METHOD PUBLIC Pop : T_PTR_STRUCT
// Remove a paper from the buffer
VAR_INPUT
END_VAR
Pop.eStatus := E_PTR_Status.Gone;
Pop.lrePositionOnBelt_mm := 0.0;
Pop.lrePositionOnBeltAdjusted_mm := 0.0;
Pop.udiItemId := 0;
Pop.udiTimeOnBelt_us := 0;


IF m_intPaperOnBelt > 0 THEN
	Pop := m_arBuffer[m_intFirstPaperIdx];
	m_arBuffer[m_intFirstPaperIdx].udiItemId := 0;
	m_arBuffer[m_intFirstPaperIdx].lrePositionOnBelt_mm := 0.0;
	m_arBuffer[m_intFirstPaperIdx].lrePositionOnBeltAdjusted_mm := 0.0;
	m_arBuffer[m_intFirstPaperIdx].udiTimeOnBelt_us := 0;
	m_arBuffer[m_intFirstPaperIdx].eStatus := E_PTR_Status.Gone;
	m_intPaperOnBelt := m_intPaperOnBelt - 1;

	IF m_intPaperOnBelt = 0 THEN
		m_arPositionList[0] := m_arBuffer[m_intFirstPaperIdx];
	END_IF

	m_intFirstPaperIdx := (m_intFirstPaperIdx + 1) MOD THIS^.cMAXBUFFERSIZE;
END_IF
END_METHOD

PROPERTY PUBLIC PositionList : POINTER TO T_PTR_STRUCT
GET
VAR
	iIdx			: INT;
	iNdx			: INT;
END_VAR
PositionList := ADR(m_arPositionList);
END_GET
SET
END_SET
END_PROPERTY

METHOD PUBLIC Push : BOOL
// Add (Push) a paper into the buffer
// Return an ID for the paper
VAR_INPUT
	In_udiItemId			: UDINT;
END_VAR
Push := FALSE;

IF m_intPaperOnBelt < THIS^.cMAXBUFFERSIZE THEN
	m_intLastPaperIdx := (m_intLastPaperIdx + 1) MOD THIS^.cMAXBUFFERSIZE;
	m_arBuffer[m_intLastPaperIdx].udiItemId := In_udiItemId;
	m_arBuffer[m_intLastPaperIdx].lrePositionOnBelt_mm := 0.0;
	m_arBuffer[m_intLastPaperIdx].lrePositionOnBeltAdjusted_mm := 0.0;
	m_arBuffer[m_intLastPaperIdx].udiTimeOnBelt_us := 0;
	m_arBuffer[m_intLastPaperIdx].eStatus := E_PTR_Status.EnterBusy;
	m_intPaperOnBelt := m_intPaperOnBelt + 1;
	Push := TRUE;
END_IF
END_METHOD

METHOD PUBLIC Reset : BOOL
VAR_INPUT
END_VAR
m_intFirstPaperIdx := 0;
m_intLastPaperIdx := -1;
m_intPaperOnBelt := 0;
END_METHOD

PROPERTY PUBLIC TimeBase : UDINT
GET
TimeBase := m_udiTimeBase_us;
END_GET
SET
m_udiTimeBase_us := TimeBase;
END_SET
END_PROPERTY

END_FUNCTION_BLOCK

// POUs/Controller/Driver/TCP (TCP communication driver)/FB_TCP
FUNCTION_BLOCK FB_TCP EXTENDS FB_CtrlBase
VAR
	/// Specific interface struct for public access
	SIf: T_Ctrl_SIf_TCP;
	intSendState: INT := 0;
	fbClientConnection: TC2_TCPIP.FB_ClientServerConnection;
	fbSend: TC2_TCPIP.FB_SocketSend;
	fbRecieve: TC2_TCPIP.FB_SocketReceive;
	/// buffer for recieved messages
	fbRecieveBuffer: FB_DataSetFifo;
	/// buffer for messages to be sendt
	fbSendBuffer: FB_DataSetFifo;
	stNextHead: ST_Header;
	bRecievedAck: BOOL;
	bRecievedNack: BOOL;
	iSendSize: UDINT;
	iNumSendTry: INT;
	tonSendTime: TON;
	pSendHeader: POINTER TO ST_Header;
	pByteSend: POINTER TO ARRAY[0..MAX_DATASET_SIZE] OF BYTE;
	pRecieveHead: POINTER TO ST_Header;
	pByteReceive: POINTER TO ARRAY[0..MAX_DATASET_SIZE] OF BYTE;
	naRecieveData: ARRAY[0..MAX_DATASET_SIZE] OF BYTE;
	pRecieveData: POINTER TO ARRAY[0..MAX_DATASET_SIZE] OF BYTE;
END_VAR
VAR CONSTANT
	cSendIdle: INT := 0;
	cSendBusy: INT := 1;
	cSendWait: INT := 2;
END_VAR

(*__________________________________________________________________________________________________
¦	
¦	Vistaprint Schweiz GmbH
¦	CH - 8401 Winterthur
¦
¦	www.vistaprint.ch - info@vistaprint.ch
¦___________________________________________________________________________________________________

Function desription:



History:
Version		Date			Author		Comment
---------------------------------------------------------------------------------------------------
0.00.1		21.05.2014		AVME/DSC	Start history. Based on TCP client from jetter prototyp (Sonja Segmueller)
___________________________________________________________________________________________________*)


SUPER^();

{attribute 'object_name' := 'Always'}
METHOD PROTECTED Always : BOOL
// not inherite from base !!!  special behaviour for this TCP driver
// SUPER^.Always();

// Conditions Always
IF (me.bolChangeBackToAUTO=TRUE) THEN // switch mode to automatic switch off controller
	//me.StateMachine.intStateNext := cSTA_OFFBusy;
	me.bolChangeBackToAUTO := FALSE;
END_IF

IF (CIf.SwCfg.bolExist=FALSE) THEN // hardware of controller does not exist
	me.StateMachine.intStateNext := cSTA_SINGLE_ANSWER;
ELSE
	;
END_IF

// ----------------------------------------------------------------------------------
// cyclic actions outside of statemachine
IF (me.StateMachine.intState<>cSTA_SINGLE_ANSWER) THEN
	
	// Cyclic call of the client connection
	fbClientConnection();	
END_IF
END_METHOD

{attribute 'object_name' := 'CtrlInit'}
METHOD CtrlInit : BOOL
// one time first cyclic call
// The socket is closed
SUPER^.CtrlInit();

me.StateMachine.intStateNext := TCP_CmdState.cSTA_Close;
END_METHOD

PROPERTY PUBLIC CtrlSIf : POINTER TO T_Ctrl_SIf_TCP
GET
CtrlSIf := ADR(SIf);
END_GET
END_PROPERTY

{attribute 'object_name' := 'CycleEndDuty'}
METHOD PROTECTED CycleEndDuty : BOOL
VAR
	intI: INT;
END_VAR
SUPER^.CycleEndDuty();

// Handle Send Data
CASE intSendState OF
	cSendIdle: 
		IF fbSendBuffer.nCount > 0 AND NOT (fbSend.bBusy) AND (fbClientConnection.eState = TC2_TCPIP.E_SocketConnectionState.eSOCKET_CONNECTED) THEN // there is something in the buffer that needs to be sent
			intSendState := cSendBusy;
			
			// Remove data from buffer. Get next package.
			fbSendBuffer.A_Remove(pHeader => pSendHeader);
			pByteSend := pSendHeader;
			stNextHead := pSendHeader^;
			
			IF (stNextHead.uinMsgId = 999) OR (stNextHead.uinMsgId = 998 ) THEN // ack or nack
				iSendSize := SIZEOF(stNextHead.uinMsgId);
			ELSE
				iSendSize := stNextHead.udiMsgSize + SIZEOF(ST_Header);
			END_IF
			
			// send Command
			fbSend(bExecute := FALSE, sSrvNetId := ''); 
			fbSend.sSrvNetId := ''; // SIf.Par.strIPAdr;
			fbSend.hSocket := fbClientConnection.hSocket;
			fbSend.cbLen := iSendSize;
			fbSend.pSrc := pByteSend;
			fbSend.bExecute := TRUE;
			fbSend.tTimeout := SIf.Par.tTOSend;
			fbSend(); 
		ELSE
			fbSend.bExecute := FALSE;
			fbSend.sSrvNetId := '';
			fbSend();
		END_IF	
		// *)
	cSendBusy:
		IF NOT (fbSend.bBusy) THEN // sending done
			
			// First Check about FUB error	
			IF (fbSend.bError = TRUE) THEN
				IF NOT (SIf.Cur.bolFubErrorActive) THEN
					SIf.Cur.bolFubErrorActive:= TRUE;																				
					pfbAlarmCtrl^.setAlarm(CIf.Info.intCtrlId,E_ALM_TCP.FubErrorSendData, UDINT_TO_DINT(fbSend.nErrId),ADR(SIf.Alm),E_AlmState.RST,CIf.Job.eMe_ActivAlmClass);																						
					// Try to close the socket. Needs reconnect for socket after an error!	
					me.StateMachine.intStateNext := TCP_CmdState.cSTA_CloseBusy;					
				END_IF	
			// no error			
			ELSE
				IF (stNextHead.uinMsgId > 997) OR (NOT (SIf.Cfg.bUsingAck)) THEN // the sent was ack or nack
					intSendState := cSendIdle;
				ELSE // wair for ack
					intSendState := cSendWait;
					tonSendTime(IN := 0);
					tonSendTime.PT := SIf.Par.iMaxWaitTimeAck;
					tonSendTime(IN := 1);
				END_IF	
			END_IF
			
		END_IF
		
		fbSend.bExecute := FALSE;
		fbSend.sSrvNetId := '';
		fbSend(); // *)
		
	cSendWait:
		fbSend.bExecute := FALSE;
		fbSend.sSrvNetId := '';
		fbSend();
		tonSendTime(IN := 1);
		// Wait for the ACK
		IF bRecievedAck THEN
			bRecievedAck := 0;
			iNumSendTry := 0; // reset for next send
			intSendState := cSendIdle;
			
		ELSIF (tonSendTime.Q) OR (bRecievedNack) THEN // timeout
			
			iNumSendTry := iNumSendTry +1;
			IF iNumSendTry >= SIf.Par.iMaxSendTry THEN
				// the signal has not been acknoledged too many times => error
				pfbAlarmCtrl^.setAlarm(CIf.Info.intCtrlId,E_ALM_TCP.NoAckRecieved,0,ADR(SIf.Alm),E_AlmState.RST,CIf.Job.eMe_ActivAlmClass);
				me.StateMachine.intStateNext := BASE_PLC.cSTA_ERROR;
			ELSE // retry sending
				fbSend.bExecute := TRUE;
				fbSend(); 
				intSendState := cSendBusy;
			END_IF
			
		END_IF
END_CASE // *)
fbSend();
END_METHOD

{attribute 'object_name' := 'CycleStartDuty'}
METHOD PROTECTED CycleStartDuty : BOOL
VAR
	bSuccess: BOOL;
	nLoad: UDINT;
	stACK: ST_Header;
END_VAR
SUPER^.CycleStartDuty();

// recieve data if connected
IF (fbClientConnection.eState = TC2_TCPIP.E_SocketConnectionState.eSOCKET_CONNECTED) THEN
	
	IF fbRecieve.bBusy THEN	
		fbRecieve.bExecute := FALSE;
		fbRecieve.sSrvNetId := '';
		fbRecieve();
		
		IF NOT (fbRecieve.bBusy) THEN
			// Recieve is finished => see what we got
				
			// First Check about FUB error	
			IF (fbRecieve.bError = TRUE) THEN
				IF NOT (SIf.Cur.bolFubErrorActive) THEN
					SIf.Cur.bolFubErrorActive:= TRUE;																				
					pfbAlarmCtrl^.setAlarm(CIf.Info.intCtrlId,E_ALM_TCP.FubErrorReceiveData, UDINT_TO_DINT(fbRecieve.nErrId),ADR(SIf.Alm),E_AlmState.RST,CIf.Job.eMe_ActivAlmClass);																						
					// Try to close the socket. Needs reconnect for socket after an error!	
					me.StateMachine.intStateNext := TCP_CmdState.cSTA_CloseBusy;					
				END_IF	
				
			// No error			
			ELSE
				// Check received data
				CASE pRecieveHead^.uinMsgId  OF
					// ACK
					// **************************
					999: 
						bRecievedAck := 1;
					
					// NACK
					// **************************
					998: 
						bRecievedNack := 1;
						
					// Valid message IDs
					// **************************
					2, 3, 4, 5, 6, 7: 
					
						fbRecieveBuffer.A_Add(in := ADR(naRecieveData), iAddSize:= UDINT_TO_INT(SIZEOF(ST_Header) + pRecieveHead^.udiMsgSize), bOk=>bSuccess , nLoad => nLoad );
						IF NOT ( bSuccess ) THEN 
							pfbAlarmCtrl^.setAlarm(CIf.Info.intCtrlId,E_ALM_TCP.AddToReceiveBufferFailed,0,ADR(SIf.Alm),E_AlmState.RST,CIf.Job.eMe_ActivAlmClass);
							me.StateMachine.intStateNext := BASE_PLC.cSTA_ERROR;
							me.StateMachine.intState := BASE_PLC.cSTA_ERROR;
						END_IF
								
					// nothing has been recieved	
					// **************************
					0: 
					
				ELSE
					// send NACK Command
					IF(SIf.Cfg.bUsingAck) THEN
						stACK.uinMsgId := 998;
						fbSendBuffer.A_Add(in := ADR(stACK), bOk=>bSuccess , nLoad => nLoad, iAddSize:= SIZEOF(stACK.uinMsgId) );
						IF NOT (bSuccess) THEN 
							pfbAlarmCtrl^.setAlarm(CIf.Info.intCtrlId,E_ALM_TCP.AddToSendBufferFailed,0,ADR(SIf.Alm),E_AlmState.RST,CIf.Job.eMe_ActivAlmClass);
							me.StateMachine.intStateNext := BASE_PLC.cSTA_ERROR;
							me.StateMachine.intState := BASE_PLC.cSTA_ERROR;
						END_IF
					END_IF
				
				END_CASE
				// empty the recieve data
				pRecieveHead^.uinMsgId := 0;			
			END_IF	
			
		END_IF
		
	// Trigger the next data receive 
	ELSE
		fbRecieve(bExecute := FALSE); // Needs new trigger!
		fbRecieve.sSrvNetId := '';
		fbRecieve.hSocket := fbClientConnection.hSocket;
		fbRecieve.cbLen := SIZEOF(naRecieveData);
		fbRecieve.pDest := ADR(naRecieveData);
		fbRecieve.tTimeout := SIf.Par.tTOReceive;
		fbRecieve.bExecute := TRUE;
		fbRecieve();
	END_IF
END_IF 
fbRecieve();
END_METHOD

{attribute 'object_name' := 'FB_init'}
METHOD FB_init : BOOL
VAR_INPUT
	/// if TRUE, the retain variables are initialized (warm start / cold start)
	bInitRetains: BOOL;
	/// if TRUE, the instance afterwards gets moved into the copy code (online change)
	bInCopyCode: BOOL;
END_VAR
VAR
	iIdx: UINT;
	iLength: UINT;
END_VAR
// ------------------------------------------------------------------------------------------------------------------------
// to manually change in new FUB implementation!!!
// define valid commands for this controller
iLength := SIZEOF(CIf.Job.aCmdList)/SIZEOF(CIf.Job.aCmdList[0]);
iIdx := 0;

WHILE (iIdx < iLength) AND (CIf.Job.aCmdList[iIdx].intCmd <> cCMD_INITIALIZED) DO
	iIdx := iIdx + 1; 
END_WHILE

IF (iIdx < iLength) THEN
// Add configuration of own comands	
	CIf.Job.aCmdList[iIdx].intCmd := TCP_CmdState.cCMD_Close;
	CIf.Job.aCmdList[iIdx].strName := 'CLOSE'; 
	CIf.Job.aCmdList[iIdx].bolAvailable := TRUE;
    iIdx := iIdx + 1;
		CIf.Job.aCmdList[iIdx].intCmd := TCP_CmdState.cCMD_Connect;
	CIf.Job.aCmdList[iIdx].strName := 'CONNECT'; 
	CIf.Job.aCmdList[iIdx].bolAvailable := TRUE;
    iIdx := iIdx + 1;

ELSE
	// Error if the aCmdList Array is to small
END_IF

// set name of class/typ
CIf.Info.strType := 'FB_TCP';
CIf.Info.strFullName := 'TCP Communication Driver';

// set alarm class
SIf.Alm[E_ALM_TCP.AddToReceiveBufferFailed].eAlmClass := E_AlmClass.INFO;
SIf.Alm[E_ALM_TCP.AddToReceiveBufferFailed].strText := 'addRecieveBufferFailed'; 
SIf.Alm[E_ALM_TCP.AddToSendBufferFailed].eAlmClass := E_AlmClass.INFO;
SIf.Alm[E_ALM_TCP.AddToSendBufferFailed].strText := 'addSendBufferFailed'; 
SIf.Alm[E_ALM_TCP.GetFromReceiveBufferFailed].eAlmClass := E_AlmClass.INFO;
SIf.Alm[E_ALM_TCP.GetFromReceiveBufferFailed].strText := 'getRecieveBufferFailed'; 
SIf.Alm[E_ALM_TCP.GetFromSendBufferFailed].eAlmClass := E_AlmClass.INFO;
SIf.Alm[E_ALM_TCP.GetFromSendBufferFailed].strText := 'getSendBufferFailed'; 
SIf.Alm[E_ALM_TCP.RemoveFromReceiveBufferFailed].eAlmClass := E_AlmClass.INFO;
SIf.Alm[E_ALM_TCP.RemoveFromReceiveBufferFailed].strText := 'RemoveRecieveBufferFailed'; 
SIf.Alm[E_ALM_TCP.RemoveFromSendBufferFailed].eAlmClass := E_AlmClass.INFO;
SIf.Alm[E_ALM_TCP.RemoveFromSendBufferFailed].strText := 'RemoveSendBufferFailed'; 
SIf.Alm[E_ALM_TCP.SocketConnectionLost].eAlmClass := E_AlmClass.INFO;
SIf.Alm[E_ALM_TCP.SocketConnectionLost].strText := 'SocketLost'; 
SIf.Alm[E_ALM_TCP.NotSent].eAlmClass := BASE_PLC.E_AlmClass.INFO;
SIf.Alm[E_ALM_TCP.NotSent].strText := 'NotSent';
SIf.Alm[E_ALM_TCP.NoAckRecieved].eAlmClass := BASE_PLC.E_AlmClass.INFO;
SIf.Alm[E_ALM_TCP.NoAckRecieved].strText := 'NoAckRecieved';
SIf.Alm[E_ALM_TCP.FubErrorClientConnection].eAlmClass := BASE_PLC.E_AlmClass.INFO;
SIf.Alm[E_ALM_TCP.FubErrorClientConnection].strText := 'FUB error - client connection. Note add. info number';
SIf.Alm[E_ALM_TCP.FubErrorSendData].eAlmClass := BASE_PLC.E_AlmClass.INFO;
SIf.Alm[E_ALM_TCP.FubErrorSendData].strText := 'FUB error - send data. Note add. info number';
SIf.Alm[E_ALM_TCP.FubErrorReceiveData].eAlmClass := BASE_PLC.E_AlmClass.INFO;
SIf.Alm[E_ALM_TCP.FubErrorReceiveData].strText := 'FUB error - receive data. Note add. info number';


// *******************************************************************************
// initial values
// *******************************************************************************

// software configuration
CIf.SwCfg.bolExist := TRUE;
CIf.SwCfg.bolEnable := TRUE;
CIf.SwCfg.bolSimulation :=  FALSE;

// parameter
SIF.Par.strIPAdr := '192.168.2.182'; 
SIF.Par.udiPort := 7443;
SIF.Par.tTOConnection := T#10S;
SIF.Par.tTOReceive := T#5S;
SIF.Par.tTOSend := T#5S;
SIf.Par.iMaxWaitTimeAck := T#4S; // wait for Ack before declaring it not recieved
SIf.Par.iMaxSendTry := 5;

SIf.Cfg.bUsingAck := TRUE;

pRecieveData := ADR(naRecieveData);
pRecieveHead := pRecieveData;
END_METHOD

{attribute 'object_name' := 'getCmdState'}
METHOD PROTECTED getCmdState : STRING
VAR_INPUT
	intCmdState: INT;
	bolState: BOOL;
END_VAR
getCmdState := SUPER^.getCmdState(intCmdState:=intCmdState,bolState:=bolState); // get global/base defined cmds/states

IF (getCmdState='') THEN // global not defined get local
	// get string cmd/state string information in runtime	
	IF (bolState=FALSE) THEN
		// States's
		CASE intCmdState OF
			TCP_CmdState.cCMD_Connect: 
				getCmdState := 'cCMD_CONNECT';
			TCP_CmdState.cCMD_Close: 
				getCmdState := 'cCMD_CLOSE';

		END_CASE;
	ELSE
		// States's
		CASE intCmdState OF
			TCP_CmdState.cSTA_Close: 
				getCmdState := 'cSTA_CLOSE';
			TCP_CmdState.cSTA_CloseBusy: 
				getCmdState := 'cSTA_CLOSEBusy';
			TCP_CmdState.cSTA_Connect: 
				getCmdState := 'cSTA_CONNECT';
			TCP_CmdState.cSTA_ConnectBusy: 
				getCmdState := 'cSTA_CONNECTBusy';			
		END_CASE;
	END_IF 
END_IF
END_METHOD

{attribute 'object_name' := 'getCtrlSIf'}
METHOD getCtrlSIf : POINTER TO T_Ctrl_SIf_TCP
getCtrlSIf := ADR(SIf);
END_METHOD

{attribute 'object_name' := 'M_Pop'}
METHOD M_Pop : BOOL
VAR_OUTPUT
	naPopMsg: ARRAY[0..MAX_DATASET_SIZE] OF BYTE;
	bPop: BOOL;
END_VAR
IF fbRecieveBuffer.nCount > 0 THEN // there is something in the recieve buffer
	fbRecieveBuffer.A_Remove( pHeader => pByteReceive );
	naPopMsg := pByteReceive^;
	M_Pop := 1;
	bPop := 1;
ELSE
	M_Pop := 0;
	bPop := 0;
END_IF
END_METHOD

{attribute 'object_name' := 'M_Push'}
METHOD M_Push : BOOL
VAR_INPUT
	paPushMsg: POINTER TO ARRAY[0..MAX_DATASET_SIZE] OF BYTE;
END_VAR
VAR
	pstPushMsg: POINTER TO ST_Header;
END_VAR
// send if desired
pstPushMsg := paPushMsg;
	
fbSendBuffer.A_Add(in := paPushMsg, iAddSize := UDINT_TO_INT(pstPushMsg^.udiMsgSize + SIZEOF(ST_HEADER)) , bOk=>M_Push );

IF NOT ( M_Push ) THEN 
	pfbAlarmCtrl^.setAlarm(CIf.Info.intCtrlId,E_ALM_TCP.AddToSendBufferFailed,0,ADR(SIf.Alm),E_AlmState.RST,CIf.Job.eMe_ActivAlmClass);
	me.StateMachine.intStateNext := BASE_PLC.cSTA_ERROR;
END_IF
END_METHOD

{attribute 'object_name' := 'sta_CLOSE'}
METHOD sta_CLOSE : BOOL
// state implemetation
// --------------------------------------------------------------------------------------
// Entry action
	IF (me.StateMachine.intState<>me.StateMachine.intStateLastCycle) THEN
		me.StateMachine.intStateLastCycle := me.StateMachine.intState;
		;
		
	END_IF

// --------------------------------------------------------------------------------------
// Cyclic action
	IF (me.StateMachine.intState=me.StateMachine.intStateLastCycle) THEN
		CASE me.intCmd OF
			TCP_CmdState.cCMD_Connect:
				me.StateMachine.intStateNext := TCP_CmdState.cSTA_ConnectBusy;
		END_CASE
	END_IF

// --------------------------------------------------------------------------------------
// Exit action
	IF (me.StateMachine.intState<>me.StateMachine.intStateNext) THEN
		;
	END_IF
END_METHOD

{attribute 'object_name' := 'sta_CLOSEBusy'}
METHOD sta_CLOSEBusy : BOOL
// state implemetation
// --------------------------------------------------------------------------------------
// Entry action
	IF (me.StateMachine.intState<>me.StateMachine.intStateLastCycle) THEN
		me.StateMachine.intStateLastCycle := me.StateMachine.intState;
		
		// Reset Tx state
		intSendState:= cSendIdle;
		fbSend.bExecute:= FALSE;
		fbRecieve.bExecute:= FALSE;
		iNumSendTry := 0;
		
		// Close socket
		fbClientConnection.bEnable:= FALSE;
		
		// clear both buffers
		fbSendBuffer.A_Reset();
		fbRecieveBuffer.A_Reset();
	END_IF

// --------------------------------------------------------------------------------------
// Cyclic action
	IF (me.StateMachine.intState=me.StateMachine.intStateLastCycle) THEN
		
		// Check about FUB error	
		IF (fbClientConnection.bError = TRUE) OR (fbClientConnection.nErrId <> 0) THEN
			SIf.Cur.bolFubErrorActive:= TRUE;																					
			pfbAlarmCtrl^.setAlarm(CIf.Info.intCtrlId,E_ALM_TCP.FubErrorClientConnection, UDINT_TO_DINT(fbClientConnection.nErrId),ADR(SIf.Alm),E_AlmState.RST,CIf.Job.eMe_ActivAlmClass);																			
			me.StateMachine.intStateNext := BASE_PLC.cSTA_ERROR;	
		END_IF
					
		// Wait until socket is closed	
		IF (fbClientConnection.eState = TC2_TCPIP.E_SocketConnectionState.eSOCKET_DISCONNECTED) THEN 	
			me.StateMachine.intStateNext := TCP_CmdState.cSTA_Close;
		ELSIF (SIf.Cur.bolFubErrorActive) THEN
			me.StateMachine.intStateNext := BASE_PLC.cSTA_ERROR;	
		END_IF
		
	END_IF
	
// --------------------------------------------------------------------------------------
// Exit action
	IF (me.StateMachine.intState<>me.StateMachine.intStateNext) THEN
		;
	END_IF
END_METHOD

{attribute 'object_name' := 'sta_CONNECT'}
METHOD sta_CONNECT : BOOL
// state implemetation
// --------------------------------------------------------------------------------------
// Entry action
	IF (me.StateMachine.intState<>me.StateMachine.intStateLastCycle) THEN
		me.StateMachine.intStateLastCycle := me.StateMachine.intState;
		;
	END_IF

// --------------------------------------------------------------------------------------
// Cyclic action
	IF (me.StateMachine.intState=me.StateMachine.intStateLastCycle) THEN

		// check if connection has been lost
		IF (fbClientConnection.eState <> TC2_TCPIP.E_SocketConnectionState.eSOCKET_CONNECTED) THEN 
			pfbAlarmCtrl^.setAlarm(CIf.Info.intCtrlId,E_ALM_TCP.SocketConnectionLost,0,ADR(SIf.Alm),E_AlmState.RST,CIf.Job.eMe_ActivAlmClass);
			me.StateMachine.intStateNext := BASE_PLC.cSTA_ERROR;
		END_IF
		
		CASE me.intCmd OF
			TCP_CmdState.cCMD_Close:
				me.StateMachine.intStateNext := TCP_CmdState.cSTA_CloseBusy;
		END_CASE
	END_IF

// --------------------------------------------------------------------------------------
// Exit action
	IF (me.StateMachine.intState<>me.StateMachine.intStateNext) THEN
		;
	END_IF
END_METHOD

{attribute 'object_name' := 'sta_CONNECTBusy'}
METHOD sta_CONNECTBusy : BOOL
// state implemetation
// --------------------------------------------------------------------------------------
// Entry action
	IF (me.StateMachine.intState<>me.StateMachine.intStateLastCycle) THEN
		me.StateMachine.intStateLastCycle := me.StateMachine.intState;
		
		// Initialize and connect socket
		fbClientConnection.nMode := 0; 	// not used
		fbClientConnection.sRemoteHost := SIf.Par.strIPAdr;
		fbClientConnection.nRemotePort := SIf.Par.udiPort;
		fbClientConnection.tReconnect := SIF.Par.tTOConnection;
		fbClientConnection.bEnable:= TRUE;
	
		// clear both buffers
		fbSendBuffer.A_Reset();
		fbRecieveBuffer.A_Reset();
		
		// reset all nessecary parameters
		bRecievedAck := 0;
		bRecievedNack := 0;
		intSendState := 0;
	END_IF


// --------------------------------------------------------------------------------------
// Cyclic action
	IF (me.StateMachine.intState=me.StateMachine.intStateLastCycle) THEN
		
		// Check about FUB error	
		IF (fbClientConnection.bError = TRUE) OR (fbClientConnection.nErrId <> 0) THEN		
			SIf.Cur.bolFubErrorActive:= TRUE;																			
			pfbAlarmCtrl^.setAlarm(CIf.Info.intCtrlId,E_ALM_TCP.FubErrorClientConnection, UDINT_TO_DINT(fbClientConnection.nErrId),ADR(SIf.Alm),E_AlmState.RST,CIf.Job.eMe_ActivAlmClass);																			
			me.StateMachine.intStateNext := BASE_PLC.cSTA_ERROR;	
		END_IF
				
		// Wait for socket handle ID and connection state
		IF (fbClientConnection.hSocket.handle <> 0) AND (fbClientConnection.eState = TC2_TCPIP.E_SocketConnectionState.eSOCKET_CONNECTED) THEN 	
			me.StateMachine.intStateNext := TCP_CmdState.cSTA_Connect;
		END_IF
		
	END_IF

// --------------------------------------------------------------------------------------
// Exit action
	IF (me.StateMachine.intState<>me.StateMachine.intStateNext) THEN
		;
	END_IF
END_METHOD

{attribute 'object_name' := 'sta_ERROR'}
METHOD PROTECTED sta_ERROR : BOOL
// state implemetation
// --------------------------------------------------------------------------------------
// Entry action
	IF (me.StateMachine.intState<>me.StateMachine.intStateLastCycle) THEN
		me.StateMachine.intStateHistory := me.StateMachine.intStateLastCycle; // -> possibillity to go back to state before error
		me.StateMachine.intStateLastCycle := me.StateMachine.intState;
		
		// Clear pending commands
		CIf.Job.intACmd:= Base_PLC.cCMD_DONE;
		CIf.Job.intMCmd:= Base_PLC.cCMD_DONE;
			
		iNumSendTry := 0;
				
		// clear both buffers
		fbSendBuffer.A_Reset();
		fbRecieveBuffer.A_Reset();
		// Reset Tx state
		intSendState:= cSendIdle;
	END_IF
	

// --------------------------------------------------------------------------------------
// Cyclic action
	IF (me.StateMachine.intState=me.StateMachine.intStateLastCycle) THEN
		
		// State Change Condition
		IF (CIf.Job.bolAlmReset = TRUE) THEN
			SIf.Cur.bolFubErrorActive:= FALSE;
			me.StateMachine.intStateNext := cSTA_ERRORQuit;
		END_IF
	END_IF

// --------------------------------------------------------------------------------------
// Exit action
	IF (me.StateMachine.intState<>me.StateMachine.intStateNext) THEN
		;
	END_IF
END_METHOD

{attribute 'object_name' := 'sta_ERRORQuit'}
METHOD PROTECTED sta_ERRORQuit : BOOL
// state implemetation
// --------------------------------------------------------------------------------------
// Entry action
	IF (me.StateMachine.intState<>me.StateMachine.intStateLastCycle) THEN
		me.StateMachine.intStateLastCycle := me.StateMachine.intState;
		;
	END_IF

// -------------------------------------------------------------------------------------
// Cyclic action
	IF (me.StateMachine.intState=me.StateMachine.intStateLastCycle) THEN
		
		IF (CIf.Job.bolAlmReset = TRUE) THEN
			CIf.Job.eMe_ActivAlmClass := E_AlmClass.NONE; // reset feedback channel for parent
			CIf.Job.bolAlmReset := FALSE;
		END_IF
		
		// State Change Condition
		IF (CIf.Job.bolAlmReset = FALSE) THEN
			// Needs reconnect for socket after an error!	
			me.StateMachine.intStateNext := TCP_CmdState.cSTA_CloseBusy;
		END_IF
	END_IF

// --------------------------------------------------------------------------------------
// Exit action
	IF (me.StateMachine.intState<>me.StateMachine.intStateNext) THEN
		;
	END_IF
END_METHOD

{attribute 'object_name' := 'StateMachine'}
METHOD PROTECTED StateMachine : BOOL
SUPER^.StateMachine();

// main statemachine of base controller
CASE me.StateMachine.intState OF
	TCP_CmdState.cSTA_Close:
		THIS^.sta_CLOSE();
    TCP_CmdState.cSTA_ConnectBusy:
		THIS^.sta_CONNECTBusy();
	TCP_CmdState.cSTA_Connect:
		THIS^.sta_CONNECT();
	TCP_CmdState.cSTA_CloseBusy:
		THIS^.sta_CLOSEBusy();
END_CASE;
END_METHOD

END_FUNCTION_BLOCK

// POUs/Controller/Utility/FiFo/FB_DataSetFifo
FUNCTION_BLOCK FB_DataSetFifo
VAR_INPUT
	bOverwrite: BOOL;
	in: POINTER TO BYTE;
	iAddSize: INT;
END_VAR
VAR_OUTPUT
	bOk: BOOL;
	nCount: UDINT;
	nLoad: UDINT;
	out: ARRAY[0..MAX_DATASET_SIZE] OF BYTE;
	pHeader: POINTER TO ST_Header;
END_VAR
VAR
	/// Buffer memory used by FB_MemRingBuffer function block 
	arrBuffer: ARRAY[0..MAX_BUFFER_SIZE] OF BYTE;
	fbBuffer: FB_MemRingBuffer;
	intLoopRemove: INT;
	intLoopReset: INT;
END_VAR
VAR CONSTANT
	MAX_BUFFER_SIZE: UDINT := 1000;
END_VAR

;

ACTION A_Add:
fbBuffer.A_AddTail( pWrite:= in,
					cbWrite:= INT_TO_UDINT(iAddSize),
					pBuffer:= ADR( arrBuffer ),
					cbBuffer:= SIZEOF( arrBuffer ),
					bOk=> bOk,
					nCount => nCount );

IF NOT bOk THEN (* overflow ? *)
	IF bOverwrite THEN
		fbBuffer.A_RemoveHead(); (* remove one oldest entry *)
		fbBuffer.A_AddTail( bOk => bOk, nCount => nCount );
	END_IF
END_IF

nLoad := (fbBuffer.cbSize * 100) / MAX_BUFFER_SIZE;
END_ACTION

ACTION A_Get:
fbBuffer.A_GetHead( pRead:= ADR( out ),
					cbRead:= SIZEOF( out ),
					pBuffer:= ADR( arrBuffer ),
					cbBuffer:= SIZEOF( arrBuffer ),
					bOk=> bOk,
					nCount => nCount );

pHeader := ADR(out);					
					
nLoad := (fbBuffer.cbSize * 100) / MAX_BUFFER_SIZE;
END_ACTION

ACTION A_Remove:
// Clean up package buffer
FOR intLoopRemove:=0 TO SIZEOF(out)-1 DO
	out[intLoopRemove]:= 0;
END_FOR

// Remove data from buffer. Get next package.
fbBuffer.A_RemoveHead( 	pRead:= ADR(out),
						cbRead:= SIZEOF(out),
						pBuffer:= ADR(arrBuffer),
						cbBuffer:= SIZEOF(arrBuffer),
						bOk=> bOk,
						nCount => nCount );
// Return						
pHeader := ADR(out);

nLoad := (fbBuffer.cbSize * 100) / MAX_BUFFER_SIZE;
END_ACTION

ACTION A_Reset:
// MEMSET not working!
//MEMSET( ADR( arrBuffer ), 0, SIZEOF( arrBuffer ) ); (* reset (optional) internal buffer *)
FOR intLoopReset:=0 TO SIZEOF(arrBuffer)-1 DO
	arrBuffer[intLoopReset]:= 0;
END_FOR

fbBuffer.A_Reset( 	bOk=> bOk,
					nCount => nCount );

nLoad := (fbBuffer.cbSize * 100) / MAX_BUFFER_SIZE;
END_ACTION

END_FUNCTION_BLOCK

// POUs/Controller/Lvl0/GRR (Granulate Remote)/helper/cycle_Grr
FUNCTION cycle_Grr : BOOL
VAR_INPUT
	pGrr: POINTER TO T_GRR;
END_VAR

pGrr^.ctrl.fbGrr.In_bolAutoMode				:= pGrr^.io.In_bolAutoMode;
pGrr^.ctrl.fbGrr.In_bolEoffOrFuseOk			:= pGrr^.io.In_bolEoffOrFuseOk;
pGrr^.ctrl.fbGrr.In_bolMainPressureError	:= pGrr^.io.In_bolMainPressureError;
pGrr^.ctrl.fbGrr.In_bolPowderLowWarning		:= pGrr^.io.In_bolPowderLowWarning;
pGrr^.ctrl.fbGrr.In_bolSystemOk				:= pGrr^.io.In_bolSystemOk;
pGrr^.ctrl.fbGrr.In_intState				:= pGrr^.io.In_intState;
pGrr^.ctrl.fbGrr.In_bolToggleBitGrn			:= pGrr^.io.In_bolToggleBitGrn;
pGrr^.ctrl.fbGrr();
pGrr^.io.Out_intCommand						:= pGrr^.ctrl.fbGrr.Out_intCommand;
pGrr^.io.Out_intConveyorBelt				:= pGrr^.ctrl.fbGrr.Out_intConveyorBelt;
pGrr^.io.Out_intConveyorVibrator			:= pGrr^.ctrl.fbGrr.Out_intConveyorVibrator;
pGrr^.io.Out_intPowderVibrator				:= pGrr^.ctrl.fbGrr.Out_intPowderVibrator;
pGrr^.io.Out_uinFilterClearingCycleTime_min	:= pGrr^.ctrl.fbGrr.Out_uinFilterClearingCycleTime_min;
pGrr^.io.Out_bolToggleBitGrr				:= pGrr^.ctrl.fbGrr.Out_bolToggleBitGrr;

END_FUNCTION

// POUs/Controller/Lvl0/GRR (Granulate Remote)/helper/init_Grr
FUNCTION init_Grr : BOOL
VAR_INPUT
	pGrr			: POINTER TO T_GRR;
	/// instance array of all controller instances
	pCtrlInst		: POINTER TO fb_CtrlBase;
	/// common interface array of all controllers (main use for PLC)
	pCtrlCIf		: POINTER TO T_Ctrl_CIf;
END_VAR

pGrr^.ctrl.fbGrr.iniAllCtrlArrays(pCtrlInst,pCtrlCIf,pGrr^.id.Grr);

END_FUNCTION

// POUs/Controller/Lvl0/GRR (Granulate Remote)/FB_GRR
FUNCTION_BLOCK FB_GRR EXTENDS FB_CtrlBase
VAR_INPUT
	In_bolSystemOk: BOOL;
	In_bolMainPressureError: BOOL;
	In_bolEoffOrFuseOk: BOOL;
	In_bolPowderLowWarning: BOOL;
	In_bolAutoMode: BOOL;
	In_intState: INT;
	In_bolToggleBitGrn: BOOL;
END_VAR
VAR_OUTPUT
	Out_intCommand: INT;
	Out_intConveyorBelt: INT;
	Out_intPowderVibrator: INT;
	Out_intConveyorVibrator: INT;
	Out_uinFilterClearingCycleTime_min: UINT;
	Out_bolToggleBitGrr: BOOL;
END_VAR
VAR
	/// Specific interface struct for public access
	SIf: T_Ctrl_SIf_Grr;
	
	udiToggleBitGrrTimer_ms		: UDINT;
	udiToggleBitGrnTimer_ms		: UDINT;
	bToggleBitGrnOld			: BOOL;
	bToggleBitOK				: BOOL;
END_VAR

(*__________________________________________________________________________________________________
¦	
¦	Vistaprint Schweiz GmbH
¦	CH - 8401 Winterthur
¦
¦	www.vistaprint.ch - info@vistaprint.ch
¦___________________________________________________________________________________________________

Function desription:

History:
Version		Date			Author		Comment
---------------------------------------------------------------------------------------------------
0.00.1		05.11.2014		BB			Start history
0.00.2		06.02.2015		BB			changed name from GRN to GRR
___________________________________________________________________________________________________*)

SUPER^();

{attribute 'object_name' := 'Always'}
METHOD PROTECTED Always : BOOL
SUPER^.Always();

// ----------------------------------------------------------------------------------
// cyclic actions outside of statemachine
IF (me.StateMachine.intState <> cSTA_SINGLE_ANSWER) THEN
	
	// Toggle Bit Grr
	udiToggleBitGrrTimer_ms := udiToggleBitGrrTimer_ms + me.FUBInfo.udiSample_ms;
	IF (udiToggleBitGrrTimer_ms > 200) THEN
		SIf.Out.bolToggleBitGrr.intern := NOT SIf.Out.bolToggleBitGrr.intern;
		udiToggleBitGrrTimer_ms := 0;
	END_IF
	
	// check Toggle Bit Grn
	udiToggleBitGrnTimer_ms := udiToggleBitGrnTimer_ms + me.FUBInfo.udiSample_ms;
	IF (SIf.In.bolToggleBitGrn.intern <> bToggleBitGrnOld) THEN
		bToggleBitGrnOld := SIf.In.bolToggleBitGrn.intern;
		udiToggleBitGrnTimer_ms := 0;
	END_IF
	bToggleBitOK := FALSE;
	IF (udiToggleBitGrnTimer_ms < 1000) THEN
		bToggleBitOK := TRUE;
	END_IF
	
	IF SIf.In.bolPowderLowWarning.intern THEN
		pfbAlarmCtrl^.setAlarm(CIf.Info.intCtrlId,E_ALM_GRR.LowPowderWarning,0,ADR(SIf.Alm),E_AlmState.RST,CIf.Job.eMe_ActivAlmClass);
	END_IF
	
	IF NOT SIf.In.bolAutoMode.intern THEN
		pfbAlarmCtrl^.setAlarm(CIf.Info.intCtrlId,E_ALM_GRR.ManualOperation,0,ADR(SIf.Alm),E_AlmState.RST,CIf.Job.eMe_ActivAlmClass);
	END_IF
	
	IF NOT bToggleBitOK THEN
		pfbAlarmCtrl^.setAlarm(CIf.Info.intCtrlId,E_ALM_GRR.LostConnection,0,ADR(SIf.Alm),E_AlmState.RST,CIf.Job.eMe_ActivAlmClass);
	END_IF
	
	// reasons are either bolMainPressureError or bolEoffOrFuseOk
	IF NOT SIf.In.bolSystemOk.intern THEN
		IF SIf.In.bolMainPressureError.intern THEN
			pfbAlarmCtrl^.setAlarm(CIf.Info.intCtrlId,E_ALM_GRR.MainPressureError,0,ADR(SIf.Alm),E_AlmState.RST,CIf.Job.eMe_ActivAlmClass);
			me.StateMachine.intStateNext := cSTA_EOFFBusy;
		ELSE
			pfbAlarmCtrl^.setAlarm(CIf.Info.intCtrlId,E_ALM_GRR.SystemError,0,ADR(SIf.Alm),E_AlmState.RST,CIf.Job.eMe_ActivAlmClass);
			me.StateMachine.intStateNext := cSTA_EOFFBusy;
		END_IF
	END_IF
	
	// set outputs
	SIf.Out.intConveyorBelt.intern := REAL_TO_INT(MAX_INT/SIf.Cfg.rMaxFreq_Hz*SIf.Par.rConveyorBelt_Hz);
	SIf.Out.intConveyorVibrator.intern := REAL_TO_INT(MAX_INT/SIf.Cfg.rMaxFreq_Hz*SIf.Par.rConveyorVibrator_Hz);
	SIf.Out.intPowderVibrator.intern := REAL_TO_INT(MAX_INT/SIf.Cfg.rMaxFreq_Hz*SIf.Par.rPowderVibrator_Hz);
	SIf.Out.uinFilterClearingCycleTime_min.intern := SIf.Par.uinFilterClearingCycleTime_min;

END_IF

// ----------------------------------------------------------------------------------
// overrule error always from base -> no EOFF State!! in EOFF go to OFF
IF (me.StateMachine.intStateNext = cSTA_EOFFBusy) THEN
	IF (me.StateMachine.intState = cSTA_OFF) THEN
		me.StateMachine.intStateNext := cSTA_OFF;
	ELSE // stay in OFF
		me.StateMachine.intStateNext := cSTA_OFFBusy;
	END_IF
END_IF
END_METHOD

PROPERTY PUBLIC CtrlSIf : POINTER TO T_Ctrl_SIf_GRR
GET
CtrlSIf := ADR(SIf);
END_GET
END_PROPERTY

{attribute 'object_name' := 'FB_init'}
METHOD FB_init : BOOL
VAR_INPUT
	/// if TRUE, the retain variables are initialized (warm start / cold start)
	bInitRetains: BOOL;
	/// if TRUE, the instance afterwards gets moved into the copy code (online change)
	bInCopyCode: BOOL;
END_VAR
VAR
	iIdx: UINT;
	iLength: UINT;
END_VAR
// ------------------------------------------------------------------------------------------------------------------------
// to manually change in new FUB implementation!!!
// define valid commands for this controller
iLength := SIZEOF(CIf.Job.aCmdList)/SIZEOF(CIf.Job.aCmdList[0]);
iIdx := 0;

WHILE (iIdx < iLength) AND (CIf.Job.aCmdList[iIdx].intCmd <> cCMD_INITIALIZED) DO
	iIdx := iIdx + 1; 
END_WHILE

IF (iIdx < iLength) THEN
// Add configuration of own comands	
	CIf.Job.aCmdList[iIdx].intCmd := BASE_PLC.cCMD_RUN;
	CIf.Job.aCmdList[iIdx].strName := 'RUN'; 
	CIf.Job.aCmdList[iIdx].bolAvailable := TRUE;
    iIdx := iIdx + 1;
ELSE
	// Error if the aCmdList Array is to small
END_IF

// set name of class/typ
CIf.Info.strType := 'FB_GRR';
CIf.Info.strFullName := 'Granulate Remote';

// set alarm class
SIf.Alm[E_ALM_GRR.SystemError].eAlmClass := E_AlmClass.OFF;
SIf.Alm[E_ALM_GRR.SystemError].strText := 'System Error';
SIf.Alm[E_ALM_GRR.MainPressureError].eAlmClass := E_AlmClass.OFF;
SIf.Alm[E_ALM_GRR.MainPressureError].strText := 'Main Pressure Error';
SIf.Alm[E_ALM_GRR.EoffOrFuseError].eAlmClass := E_AlmClass.OFF;
SIf.Alm[E_ALM_GRR.EoffOrFuseError].strText := 'Eoff or Fuse Error';
SIf.Alm[E_ALM_GRR.LowPowderWarning].eAlmClass := E_AlmClass.WARNING;
SIf.Alm[E_ALM_GRR.LowPowderWarning].strText := 'Low Powder';
SIf.Alm[E_ALM_GRR.ManualOperation].eAlmClass := E_AlmClass.WARNING;
SIf.Alm[E_ALM_GRR.ManualOperation].strText := 'Manual Operation';
SIf.Alm[E_ALM_GRR.LostConnection].eAlmClass := E_AlmClass.OFF;
SIf.Alm[E_ALM_GRR.LostConnection].strText := 'Lost Connection to the Granulate Machine';

// *******************************************************************************
// initial values
// *******************************************************************************

// software configuration
CIf.SwCfg.bolExist := TRUE;
CIf.SwCfg.bolEnable := TRUE;
CIf.SwCfg.bolSimulation :=  FALSE;

// configuration
SIf.Cfg.rMaxFreq_Hz := 50.0;

// parameter
SIf.Par.rConveyorBelt_Hz		:= SIf.Cfg.rMaxFreq_Hz/2;
SIf.Par.rConveyorVibrator_Hz	:= SIf.Cfg.rMaxFreq_Hz/2;
SIf.Par.rPowderVibrator_Hz		:= SIf.Cfg.rMaxFreq_Hz/2;
SIf.Par.uinFilterClearingCycleTime_min	:= 4*60;
END_METHOD

{attribute 'object_name' := 'getCtrlSIf'}
METHOD getCtrlSIf : POINTER TO T_Ctrl_SIf_GRR
getCtrlSIf := ADR(SIf);
END_METHOD

{attribute 'object_name' := 'IoInBridge'}
METHOD PROTECTED IoInBridge : BOOL
SUPER^.IoInBridge();
// digitale and analoge inputs read from hardware or forcing
SIf.In.bolSystemOk.map	:= THIS^.In_bolSystemOk;
SIf.In.bolMainPressureError.map	:= THIS^.In_bolMainPressureError;
SIf.In.bolEoffOrFuseOk.map	:= THIS^.In_bolEoffOrFuseOk;
SIf.In.bolPowderLowWarning.map	:= THIS^.In_bolPowderLowWarning;
SIf.In.bolAutoMode.map	:= THIS^.In_bolAutoMode;
SIf.In.intState.map	:= THIS^.In_intState;
SIf.In.bolToggleBitGrn.map	:= THIS^.In_bolToggleBitGrn;

IF (CIf.SwCfg.bolSimulation = FALSE) THEN
	BASE_PLC.getInBol(CIf.Job.bolIoForce,ADR(SIf.In.bolSystemOk));
	BASE_PLC.getInBol(CIf.Job.bolIoForce,ADR(SIf.In.bolMainPressureError));
	BASE_PLC.getInBol(CIf.Job.bolIoForce,ADR(SIf.In.bolEoffOrFuseOk));
	BASE_PLC.getInBol(CIf.Job.bolIoForce,ADR(SIf.In.bolPowderLowWarning));
	BASE_PLC.getInBol(CIf.Job.bolIoForce,ADR(SIf.In.bolAutoMode));
	BASE_PLC.getInInt(CIf.Job.bolIoForce,ADR(SIf.In.intState));
	BASE_PLC.getInBol(CIf.Job.bolIoForce,ADR(SIf.In.bolToggleBitGrn));
ELSE
	//simulation of global IO
	SIf.In.bolSystemOk.intern	:= TRUE;
	SIf.In.bolMainPressureError.intern	:= FALSE;
	SIf.In.bolEoffOrFuseOk.intern	:= TRUE;
	SIf.In.bolPowderLowWarning.intern	:= FALSE;
	SIf.In.bolAutoMode.intern	:= TRUE;
	SIf.In.intState.intern	:= SIf.Out.intCommand.intern;
	SIf.In.bolToggleBitGrn.intern	:= SIf.Out.bolToggleBitGrr.intern;
END_IF
END_METHOD

{attribute 'object_name' := 'IoOutBridge'}
METHOD PROTECTED IoOutBridge : BOOL
// digitale and analoge inputs read from hardware or forcing
IF (CIf.SwCfg.bolSimulation = FALSE) THEN
	setOutInt(CIf.Job.bolIoForce ,ADR(SIf.Out.intCommand));
	setOutInt(CIf.Job.bolIoForce ,ADR(SIf.Out.intConveyorBelt));
	setOutInt(CIf.Job.bolIoForce ,ADR(SIf.Out.intConveyorVibrator));
	setOutInt(CIf.Job.bolIoForce ,ADR(SIf.Out.intPowderVibrator));
	setOutUint(CIf.Job.bolIoForce ,ADR(SIf.Out.uinFilterClearingCycleTime_min));
	setOutBol(CIf.Job.bolIoForce ,ADR(SIf.Out.bolToggleBitGrr));
	
	THIS^.Out_intCommand := SIf.Out.intCommand.map;
	THIS^.Out_intConveyorBelt := SIf.Out.intConveyorBelt.map;
	THIS^.Out_intConveyorVibrator := SIf.Out.intConveyorVibrator.map;
	THIS^.Out_intPowderVibrator := SIf.Out.intPowderVibrator.map;
	THIS^.Out_uinFilterClearingCycleTime_min := SIf.Out.uinFilterClearingCycleTime_min.map;
	THIS^.Out_bolToggleBitGrr := SIf.Out.bolToggleBitGrr.map;
ELSE
	THIS^.Out_intCommand := 0;
	THIS^.Out_intConveyorBelt := 0;
	THIS^.Out_intConveyorVibrator := 0;
	THIS^.Out_intPowderVibrator := 0;
	THIS^.Out_uinFilterClearingCycleTime_min := 0;
	THIS^.Out_bolToggleBitGrr := SIf.Out.bolToggleBitGrr.map;
END_IF
END_METHOD

{attribute 'object_name' := 'sta_ERROR'}
METHOD PROTECTED sta_ERROR : BOOL
// state implemetation
//--------------------------------------------------------------------------------------
// Entry action
	IF (me.StateMachine.intState<>me.StateMachine.intStateLastCycle) THEN
		me.StateMachine.intStateHistory := me.StateMachine.intStateLastCycle; // -> possibillity to go back to state before error
		me.StateMachine.intStateLastCycle := me.StateMachine.intState;
		
		SIf.Out.intCommand.intern := cCMD_OFF;
	END_IF


//--------------------------------------------------------------------------------------
// Cyclic action

	// State Change Condition
	IF (CIf.Job.bolAlmReset = TRUE) THEN
		me.StateMachine.intStateNext := cSTA_ERRORQuit;
	END_IF

	
//--------------------------------------------------------------------------------------
// Exit action
	IF (me.StateMachine.intState<>me.StateMachine.intStateNext) THEN
		;
	END_IF
END_METHOD

{attribute 'object_name' := 'sta_ERRORQuit'}
METHOD PROTECTED sta_ERRORQuit : BOOL
// state implemetation
//--------------------------------------------------------------------------------------
// Entry action
	IF (me.StateMachine.intState<>me.StateMachine.intStateLastCycle) THEN
		me.StateMachine.intStateLastCycle := me.StateMachine.intState;
	END_IF


//--------------------------------------------------------------------------------------
// Cyclic action
	
	// State Change Condition
	IF (CIf.Job.bolAlmReset = FALSE) THEN
		me.StateMachine.intStateNext := cSTA_OFFBusy;
	END_IF
	

//--------------------------------------------------------------------------------------
// Exit action
	IF (me.StateMachine.intState<>me.StateMachine.intStateNext) THEN
		;
	END_IF
END_METHOD

{attribute 'object_name' := 'sta_OFF'}
METHOD PROTECTED sta_OFF : BOOL
// state implemetation
// --------------------------------------------------------------------------------------
// Entry action
	IF (me.StateMachine.intState<>me.StateMachine.intStateLastCycle) THEN
		me.StateMachine.intStateLastCycle := me.StateMachine.intState;
	END_IF


// --------------------------------------------------------------------------------------
// Cyclic action

	IF me.intCmd=Base_PLC.cCMD_RUN AND SIf.In.bolSystemOk.intern THEN
		me.StateMachine.intStateNext := Base_PLC.cSTA_RUNBusy;
	END_IF


// --------------------------------------------------------------------------------------
// Exit action
	IF (me.StateMachine.intState<>me.StateMachine.intStateNext) THEN
		;
	END_IF
END_METHOD

{attribute 'object_name' := 'sta_OFFBusy'}
METHOD PROTECTED sta_OFFBusy : BOOL
// state implemetation
// --------------------------------------------------------------------------------------
// Entry action
	IF (me.StateMachine.intState<>me.StateMachine.intStateLastCycle) THEN
		me.StateMachine.intStateLastCycle := me.StateMachine.intState;
		
		SIf.Out.intCommand.intern := cCMD_OFF;
	END_IF


// --------------------------------------------------------------------------------------
// Cyclic action

	IF (SIf.In.intState.intern=cSTA_OFF OR NOT SIf.In.bolAutoMode.intern) THEN
		me.StateMachine.intStateNext := cSTA_OFF;
	END_IF

	
// --------------------------------------------------------------------------------------
// Exit action
	IF (me.StateMachine.intState<>me.StateMachine.intStateNext) THEN
		;
	END_IF
END_METHOD

{attribute 'object_name' := 'sta_PON'}
METHOD PROTECTED sta_PON : BOOL
// state implemetation
// --------------------------------------------------------------------------------------
// Entry action
	IF (me.StateMachine.intState<>me.StateMachine.intStateLastCycle) THEN
		me.StateMachine.intStateLastCycle := me.StateMachine.intState;
	END_IF

	
// --------------------------------------------------------------------------------------
// Cyclic action

	IF me.intCmd>Base_PLC.cCMD_PON THEN				
		me.StateMachine.intStateNext := Base_PLC.cSTA_OFFBusy;
	END_IF
	
	
// --------------------------------------------------------------------------------------
// Exit action
	IF (me.StateMachine.intState<>me.StateMachine.intStateNext) THEN
		;
	END_IF
END_METHOD

{attribute 'object_name' := 'sta_PONBusy'}
METHOD PROTECTED sta_PONBusy : BOOL
// state implemetation
// --------------------------------------------------------------------------------------
// Entry action
IF (me.StateMachine.intState<>me.StateMachine.intStateLastCycle) THEN
	me.StateMachine.intStateLastCycle := me.StateMachine.intState;
	
	IF SIf.In.intState.intern<=cSTA_PON THEN
		SIf.Out.intCommand.intern := cCMD_PON;
	ELSE
		SIf.Out.intCommand.intern := cCMD_OFF;
	END_IF
END_IF


// --------------------------------------------------------------------------------------
// Cyclic action

	IF SIf.In.intState.intern=cSTA_PON OR SIf.In.intState.intern=cSTA_OFF THEN
		me.StateMachine.intStateNext := cSTA_PON;
	END_IF


// --------------------------------------------------------------------------------------
// Exit action
IF (me.StateMachine.intState<>me.StateMachine.intStateNext) THEN
	;
END_IF
END_METHOD

{attribute 'object_name' := 'sta_RUN'}
METHOD PROTECTED sta_RUN : BOOL
// state implemetation
// --------------------------------------------------------------------------------------
// Entry action
	IF (me.StateMachine.intState<>me.StateMachine.intStateLastCycle) THEN
		me.StateMachine.intStateLastCycle := me.StateMachine.intState;
	END_IF


// --------------------------------------------------------------------------------------
// Cyclic action

	IF me.intCmd=Base_PLC.cCMD_OFF THEN
		me.StateMachine.intStateNext := Base_PLC.cSTA_OFFBusy;
	END_IF


// --------------------------------------------------------------------------------------
// Exit action
	IF (me.StateMachine.intState<>me.StateMachine.intStateNext) THEN
		;
	END_IF
END_METHOD

{attribute 'object_name' := 'sta_RUNBusy'}
METHOD PROTECTED sta_RUNBusy : BOOL
// state implemetation
// --------------------------------------------------------------------------------------
// Entry action
	IF (me.StateMachine.intState<>me.StateMachine.intStateLastCycle) THEN
		me.StateMachine.intStateLastCycle := me.StateMachine.intState;
		
		SIf.Out.intCommand.intern := cCMD_RUN;
	END_IF


// --------------------------------------------------------------------------------------
// Cyclic action

	IF me.intCmd=Base_PLC.cCMD_OFF THEN
		me.StateMachine.intStateNext := Base_PLC.cSTA_OFFBusy;
	ELSIF SIf.In.intState.intern=cSTA_RUN THEN
		me.StateMachine.intStateNext := Base_PLC.cSTA_RUN;
	END_IF


// --------------------------------------------------------------------------------------
// Exit action
	IF (me.StateMachine.intState<>me.StateMachine.intStateNext) THEN
		;
	END_IF
END_METHOD

{attribute 'object_name' := 'StateMachine'}
METHOD PROTECTED StateMachine : BOOL
SUPER^.StateMachine();

// main statemachine of base controller
CASE me.StateMachine.intState OF
	cSTA_RUNBusy: 
        THIS^.sta_RUNBusy();
	cSTA_RUN: 
        THIS^.sta_RUN();
END_CASE
END_METHOD

END_FUNCTION_BLOCK

// POUs/Controller/Lvl0/JCL (Jetter Client)/helper/cycle_Jcl
FUNCTION cycle_Jcl : BOOL
VAR_INPUT
	pJcl: POINTER TO T_JCL;
END_VAR

pJcl^.ctrl.fbJcl_Tcp();

pJcl^.ctrl.fbJcl();

END_FUNCTION

// POUs/Controller/Lvl0/JCL (Jetter Client)/helper/init_Jcl
FUNCTION init_Jcl : BOOL
VAR_INPUT
	pJcl			: POINTER TO T_JCL;
	/// instance array of all controller instances
	pCtrlInst		: POINTER TO fb_CtrlBase;
	/// common interface array of all controllers (main use for PLC)
	pCtrlCIf		: POINTER TO T_Ctrl_CIf;
END_VAR

pJcl^.ctrl.fbJcl_Tcp.iniAllCtrlArrays(pCtrlInst,pCtrlCIf,pJcl^.id.Jcl_Tcp);
pJcl^.ctrl.fbJcl.iniAllCtrlArrays(pCtrlInst,pCtrlCIf,pJcl^.id.Jcl);
pJcl^.ctrl.fbJcl.TCP := ADR(pJcl^.ctrl.fbJcl_Tcp);

END_FUNCTION

// POUs/Controller/Lvl0/JCL (Jetter Client)/FB_JCL
FUNCTION_BLOCK FB_JCL EXTENDS FB_CtrlBase
VAR
	/// Specific interface struct for public access
	SIf: T_Ctrl_SIf_JCL;
	/// pointer to function block
	p_fbTCP: POINTER TO FB_TCP;
	pTCP_CIF: POINTER TO BASE_PLC.T_Ctrl_CIf;
	fbStateLookup: FB_LookupTable;
	fbCommandLookup: FB_LookupTable;
	bolServerConnectionError: BOOL;
END_VAR

(*__________________________________________________________________________________________________
¦	
¦	Vistaprint Schweiz GmbH
¦	CH - 8401 Winterthur
¦
¦	www.vistaprint.ch - info@vistaprint.ch
¦___________________________________________________________________________________________________

Function desription:
ToDo: DSC...

History:
Version		Date			Author				Comment
---------------------------------------------------------------------------------------------------
0.00.1		20.05.2014		AVME/DSC			Start history. Insert all basic functionalities.
___________________________________________________________________________________________________*)

SUPER^();

{attribute 'object_name' := 'Always'}
METHOD PROTECTED Always : BOOL
// not inherite from base !!!  special behaviour for this controller
// SUPER^.Always();

// Conditions Always
IF (me.bolChangeBackToAUTO=TRUE) THEN // switch mode to automatic switch off controller
	//me.StateMachine.intStateNext := cSTA_OFFBusy;
	me.bolChangeBackToAUTO := FALSE;
END_IF

IF (CIf.SwCfg.bolExist=FALSE) THEN // hardware of controller does not exist
	me.StateMachine.intStateNext := cSTA_SINGLE_ANSWER;
ELSE
	// Handle command PON
	IF (me.intCmd=cCMD_PON) 
		AND (me.StateMachine.intState<>cSTA_PONBusy) AND (me.StateMachine.intState<>cSTA_PON)
		AND (me.StateMachine.intState<>cSTA_ERROR) AND (me.StateMachine.intState<>cSTA_ERRORQuit) 
		AND (me.StateMachine.intState<>cSTA_EOFF) AND (me.StateMachine.intState<>cSTA_EOFFBusy) THEN
		me.StateMachine.intStateNext := cSTA_PONBusy;
	END_IF
END_IF
		
// ----------------------------------------------------------------------------------
// cyclic actions outside of statemachine
IF (me.StateMachine.intState<>cSTA_SINGLE_ANSWER) THEN
	
	// Simulation
	IF (CIf.SwCfg.bolSimulation) THEN
		;
	END_IF
	
	// Always handle recieve data from jetter server
	IF NOT CIf.SwCfg.bolSimulation THEN
		THIS^.HandleReceiveData();
	END_IF
	
	// Request state
	// ------------------------------
	IF (me.intCmd=cCMD_RequestState) THEN
		// Request state one time
		CIf.Job.intACmd := Base_PLC.cCMD_DONE;
		CIf.Job.intMCmd := Base_PLC.cCMD_DONE;
		THIS^.RequestState();
	END_IF
	
	// Reset Jetter alarms
	// ------------------------------
	// Can be done over command "cCMD_ResetAlarm" or normal global AlmReset
	IF (me.intCmd=cCMD_ResetAlarm) OR ((CIf.Job.bolAlmReset = TRUE) AND (me.StateMachine.intState<>cSTA_ERROR) AND (me.StateMachine.intState<>cSTA_ERRORQuit)) THEN
		CIf.Job.bolAlmReset := FALSE;
		IF (me.intCmd=cCMD_ResetAlarm) THEN
			CIf.Job.intACmd := Base_PLC.cCMD_DONE;
			CIf.Job.intMCmd := Base_PLC.cCMD_DONE;
		END_IF
		// Reset Jetter alarms one time
		THIS^.ResetAlarms();
	END_IF	
		
END_IF

// ----------------------------------------------------------------------------------
// Always change actions in Base Library
// ----------------------------------------------------------------------------------
// overrule error always from base -> no EOFF State!! in EOFF go to OFF
IF (me.StateMachine.intStateNext = cSTA_EOFFBusy) THEN
	IF (me.StateMachine.intState=cSTA_OFF) THEN
		me.StateMachine.intStateNext := cSTA_OFF;
	ELSE // stay in OFF
		me.StateMachine.intStateNext := cSTA_OFFBusy;
	END_IF
END_IF

// Conditions Always
IF (((me.Alarm.eActivAlmClass=E_AlmClass.EOFF) OR (me.Alarm.eActivAlmClass=E_AlmClass.OFF) OR (me.intCmd=cCMD_OFF))
		 AND (me.StateMachine.intState<>cSTA_ERROR) AND (me.StateMachine.intState<>cSTA_ERRORQuit) AND
		(me.StateMachine.intState<>cSTA_OFF) AND (me.StateMachine.intState<>cSTA_OFFBusy)) THEN
	// alarm evt EOFF, OFF or cmd off
	me.StateMachine.intStateNext := cSTA_OFFBusy;
END_IF
END_METHOD

{attribute 'object_name' := 'checkChildAlmClass'}
METHOD checkChildAlmClass : BOOL
// If there is a TCP connection problem to the server
IF (pTCP_CIF^.Job.eMe_ActivAlmClass >= E_AlmClass.TSTOP) THEN
	bolServerConnectionError:= TRUE;
	// set me alarm class OFF
	CIf.Job.eMe_ActivAlmClass := E_AlmClass.OFF;
	me.StateMachine.intStateNext := Base_PLC.cSTA_ERROR;
END_IF
END_METHOD

{attribute 'object_name' := 'CtrlInit'}
METHOD CtrlInit : BOOL
SUPER^.CtrlInit();

// one time first cyclic call!
// Open the TCP communication to jetter remote server to get the actual machine state
me.StateMachine.intStateNext := JCL_CmdState.cSTA_ConnectBusy;

// get child if
pTCP_CIF 	:= AddChild(p_fbTCP^);
END_METHOD

PROPERTY PUBLIC CtrlSIf : POINTER TO T_Ctrl_SIf_JCL
GET
CtrlSIf := ADR(SIf);
END_GET
END_PROPERTY

{attribute 'object_name' := 'FB_init'}
METHOD FB_init : BOOL
VAR_INPUT
	/// if TRUE, the retain variables are initialized (warm start / cold start)
	bInitRetains: BOOL;
	/// if TRUE, the instance afterwards gets moved into the copy code (online change)
	bInCopyCode: BOOL;
END_VAR
VAR
	iIdx: UINT;
	iLength: UINT;
END_VAR
// ------------------------------------------------------------------------------------------------------------------------
// to manually change in new FUB implementation!!!
// define valid commands for this controller
iLength := SIZEOF(CIf.Job.aCmdList)/SIZEOF(CIf.Job.aCmdList[0]);
iIdx := 0;

WHILE (iIdx < iLength) AND (CIf.Job.aCmdList[iIdx].intCmd <> cCMD_INITIALIZED) DO
	iIdx := iIdx + 1; 
END_WHILE

IF (iIdx < iLength) THEN
// Add configuration of own comands	
	CIf.Job.aCmdList[iIdx].intCmd := BASE_PLC.cCMD_RUN;
	CIf.Job.aCmdList[iIdx].strName := 'RUN'; 
	CIf.Job.aCmdList[iIdx].bolAvailable := TRUE;
    iIdx := iIdx + 1;
	CIf.Job.aCmdList[iIdx].intCmd := JCL_CmdState.cCMD_Standby;
	CIf.Job.aCmdList[iIdx].strName := 'STANDBY'; 
	CIf.Job.aCmdList[iIdx].bolAvailable := TRUE;
	iIdx := iIdx + 1;
	CIf.Job.aCmdList[iIdx].intCmd := JCL_CmdState.cCMD_CleanPrintHeads;
	CIf.Job.aCmdList[iIdx].strName := 'CLEANING'; 
	CIf.Job.aCmdList[iIdx].bolAvailable := TRUE;
	iIdx := iIdx + 1;
	CIf.Job.aCmdList[iIdx].intCmd := JCL_CmdState.cCMD_Calibration;
	CIf.Job.aCmdList[iIdx].strName := 'CALIBRATION'; 
	CIf.Job.aCmdList[iIdx].bolAvailable := TRUE;
	iIdx := iIdx + 1;
	CIf.Job.aCmdList[iIdx].intCmd := JCL_CmdState.cCMD_ResetAlarm;
	CIf.Job.aCmdList[iIdx].strName := 'RESET ALARM'; 
	CIf.Job.aCmdList[iIdx].bolAvailable := TRUE;
	iIdx := iIdx + 1;
	CIf.Job.aCmdList[iIdx].intCmd := JCL_CmdState.cCMD_RequestState;
	CIf.Job.aCmdList[iIdx].strName := 'REQUEST STATE'; 
	CIf.Job.aCmdList[iIdx].bolAvailable := TRUE;
ELSE
	// Error if the aCmdList Array is to small
END_IF

// set name of class/typ
CIf.Info.strType := 'FB_JCL';
CIf.Info.strFullName := 'Jetter Client';

// set alarm class
SIf.Alm[E_ALM_JCL.none].eAlmClass := E_AlmClass.TSTOP;
SIf.Alm[E_ALM_JCL.none].strText := ''; 


// *******************************************************************************
// initial values
// *******************************************************************************

// software configuration
CIf.SwCfg.bolExist := TRUE;
CIf.SwCfg.bolEnable := TRUE;
CIf.SwCfg.bolSimulation :=  FALSE;

// Fill the lookup table with all valid jetter states
fbStateLookup.A_Add(iAddKey := Base_PLC.cSTA_EOFFBusy, iAddValue:= 3);
fbStateLookup.A_Add(iAddKey := Base_PLC.cSTA_EOFF, iAddValue:= 4);
fbStateLookup.A_Add(iAddKey := Base_PLC.cSTA_PONBusy, iAddValue:= 1);
fbStateLookup.A_Add(iAddKey := Base_PLC.cSTA_PON, iAddValue:= 2);
fbStateLookup.A_Add(iAddKey := BASE_PLC.cSTA_OFFBusy, iAddValue:= 5);
fbStateLookup.A_Add(iAddKey := BASE_PLC.cSTA_OFF, iAddValue:= 6);
fbStateLookup.A_Add(iAddKey := JCL_CmdState.cSTA_ParkBusy, iAddValue:= 211);
fbStateLookup.A_Add(iAddKey := BASE_PLC.cSTA_INITBusy, iAddValue:= 7);
fbStateLookup.A_Add(iAddKey := BASE_PLC.cSTA_INIT, iAddValue:= 8);
fbStateLookup.A_Add(iAddKey := JCL_CmdState.cSTA_StandbyBusy, iAddValue:= 201);
fbStateLookup.A_Add(iAddKey := JCL_CmdState.cSTA_Standby, iAddValue:= 202);
fbStateLookup.A_Add(iAddKey := BASE_PLC.cSTA_RUNBusy, iAddValue:= 9);
fbStateLookup.A_Add(iAddKey := BASE_PLC.cSTA_RUN, iAddValue:= 10);
fbStateLookup.A_Add(iAddKey := JCL_CmdState.cSTA_CalibrationBusy, iAddValue:= 203);
fbStateLookup.A_Add(iAddKey := JCL_CmdState.cSTA_Calibration, iAddValue:= 204);
fbStateLookup.A_Add(iAddKey := JCL_CmdState.cSTA_CleanPrintHeadsBusy, iAddValue:= 205);
fbStateLookup.A_Add(iAddKey := JCL_CmdState.cSTA_CleanPrintHeads, iAddValue:= 206);
fbStateLookup.A_Add(iAddKey := JCL_CmdState.cSTA_MaintenanceBusy, iAddValue:= 208);
fbStateLookup.A_Add(iAddKey := JCL_CmdState.cSTA_MaintenanceInWork, iAddValue:= 209);
fbStateLookup.A_Add(iAddKey := JCL_CmdState.cSTA_MaintenanceDone, iAddValue:= 210);

// prepare to recieve data
SIf.Cur.paNextMsg := ADR(SIf.Cur.naNextMsg);
SIf.Cur.puNextMsg := SIf.Cur.paNextMsg;

SIf.Cur.bolNeedsCleaning:= FALSE;	
SIf.Cur.intJETState:= 0;  // current state not yet known
END_METHOD

{attribute 'object_name' := 'getCmdState'}
METHOD PROTECTED getCmdState : STRING
VAR_INPUT
	intCmdState: INT;
	bolState: BOOL;
END_VAR
getCmdState := SUPER^.getCmdState(intCmdState:=intCmdState,bolState:=bolState); // get global/base defined cmds/states

IF (getCmdState='') THEN // global not defined get local
	// get string cmd/state string information in runtime	
	IF (bolState=FALSE) THEN
		// States's
		CASE intCmdState OF
			JCL_CmdState.cCMD_Standby: 
				getCmdState := 'cCMD_Standby';
			JCL_CmdState.cCMD_CleanPrintHeads: 
				getCmdState := 'cCMD_CleanPrintHeads';		
				
		END_CASE;
	ELSE
		// States's
		CASE intCmdState OF			
			// Main states
			JCL_CmdState.cSTA_StandbyBusy: 
				getCmdState := 'cSTA_StandbyBusy'; 
			JCL_CmdState.cSTA_Standby:
				getCmdState := 'cSTA_Standby';			
			JCL_CmdState.cSTA_ConnectBusy:
				getCmdState := 'cSTA_ConnectBusy';
			JCL_CmdState.cSTA_CleanPrintHeadsBusy: 
				getCmdState := 'cSTA_CleanPrintHeadsBusy'; 
			JCL_CmdState.cSTA_CleanPrintHeads:
				getCmdState := 'cSTA_CleanPrintHeads';		
			JCL_CmdState.cSTA_CalibrationBusy:
				getCmdState := 'cSTA_CalibrationBusy';	
			JCL_CmdState.cSTA_Calibration:
				getCmdState := 'cSTA_Calibration';	
						
			// Sub states
			JCL_CmdState.cSUB_WaitingForConnection:
				getCmdState := 'cSUB_WaitingForConnection';
			JCL_CmdState.cSUB_WaitingForState:
				getCmdState := 'cSUB_WaitingForState';
			JCL_CmdState.cSUB_Done:
				getCmdState := 'cSUB_Done';			
		END_CASE;
	END_IF 
END_IF
END_METHOD

{attribute 'object_name' := 'getCtrlSIf'}
METHOD getCtrlSIf : POINTER TO T_Ctrl_SIf_JCL
getCtrlSIf := ADR(SIf);
END_METHOD

{attribute 'object_name' := 'HandleReceiveData'}
METHOD HandleReceiveData
VAR
	bPop: BOOL;
	ii: INT;
END_VAR
// get next message
p_fbTCP^.M_Pop(naPopMsg => SIf.Cur.naNextMsg, bPop => bPop);

IF bPop THEN // something has been recieved
	CASE SIf.Cur.puNextMsg^.State.stHeader.uinMsgId OF

		// -----------------------------------------------
		// Handle received state
		// -----------------------------------------------
		// Note: The Status is send on Request and on Status Change
		JCL_MsgId_State:
			
			// Update the main state
			fbStateLookup.A_LookupByValue(iLookupValue := SIf.Cur.puNextMsg^.State.usiMainState, iFoundKey => SIf.Cur.intJETState);
	
			// Prepare additional states
			(*
			State				BIT		Description
			-------------------------------------------------------------------------------------------------
			ReadyForProduction	0		Jetter ready for production
			Running				1		Print running, in production
			NeedsAttention		2		System needs attention. Info or warning active
			Error				3		General error active
			CleaningIncomplete	4		Cleaning cycle was aborted before finishing. Production not possible.
			 -					5	 	-
			IsLocalControlled	6		Local control active. Commands from Client are ignored
			IsRemoteControlled	7		Remote control active. Commands from Client are accepted
			*)
	
			SIf.Cur.bolReadyForProduction:= SIf.Cur.puNextMsg^.State.usiAddState.0;			
			SIf.Cur.bolRunning:= SIf.Cur.puNextMsg^.State.usiAddState.1;		
			SIf.Cur.bolNeedsAttention:= SIf.Cur.puNextMsg^.State.usiAddState.2;			
			SIf.Cur.bolError:= SIf.Cur.puNextMsg^.State.usiAddState.3;			
			SIf.Cur.bolCleaningIncomplete:= SIf.Cur.puNextMsg^.State.usiAddState.4;			
			SIf.Cur.bolIsLocalControlled:= SIf.Cur.puNextMsg^.State.usiAddState.6;		
			SIf.Cur.bolIsRemoteControlled:= SIf.Cur.puNextMsg^.State.usiAddState.7;
			
		// -----------------------------------------------
		// Handle received print info (print done)
		// -----------------------------------------------		
		JCL_MsgId_PrintDone:
			;
		
		// -----------------------------------------------
		// Handle received alarm message
		// -----------------------------------------------
		JCL_MsgId_Alarm:
			;
			
		// -----------------------------------------------
		// Handle received request for cleaning
		// -----------------------------------------------
		JCL_MsgId_ReqCleaning:
				
			SIf.Cur.bolNeedsCleaning:= TRUE;			
			SIf.Cur.strDTOfLastCleaningCycle:= SIf.Cur.puNextMsg^.ReqCleaning.strDTLastClean;
		
		// nothing received	
		0:
			; 
	ELSE
		; // To do: Add error	
	END_CASE
	
END_IF
END_METHOD

{attribute 'object_name' := 'RequestState'}
METHOD PROTECTED RequestState : BOOL
VAR
	stNextCommand: T_JCL_Command;
	pNextCommand: POINTER TO T_JCL_Command;
END_VAR
// Request jetter state
IF NOT (CIf.SwCfg.bolSimulation) THEN
	stNextCommand.stHeader.uinMsgId := JCL_MsgId_Command;
	stNextCommand.stHeader.udiMsgSize := SIZEOF(T_JCL_Command) - SIZEOF(ST_Header);
	stNextCommand.usiCommand := JCL_CMD_RequestState;
	pNextCommand := ADR(stNextCommand);	
	p_fbTCP^.M_Push(paPushMsg := pNextCommand);		
END_IF
END_METHOD

{attribute 'object_name' := 'ResetAlarms'}
METHOD PROTECTED ResetAlarms : BOOL
VAR
	stNextCommand: T_JCL_Command;
	pNextCommand: POINTER TO T_JCL_Command;
END_VAR
// Request jetter state
IF NOT (CIf.SwCfg.bolSimulation) THEN
	stNextCommand.stHeader.uinMsgId := JCL_MsgId_Command;
	stNextCommand.stHeader.udiMsgSize := SIZEOF(T_JCL_Command) - SIZEOF(ST_Header);
	stNextCommand.usiCommand := JCL_CMD_ResetAlarm;
	pNextCommand := ADR(stNextCommand);	
	p_fbTCP^.M_Push(paPushMsg := pNextCommand);		
END_IF
END_METHOD

{attribute 'object_name' := 'sta_CALIBRATION'}
METHOD PROTECTED sta_CALIBRATION : BOOL
// state implemetation
// --------------------------------------------------------------------------------------
// Entry action
	IF (me.StateMachine.intState<>me.StateMachine.intStateLastCycle) THEN
		me.StateMachine.intStateLastCycle := me.StateMachine.intState;
		;
	END_IF

// --------------------------------------------------------------------------------------
// Cyclic action
	IF (me.StateMachine.intState=me.StateMachine.intStateLastCycle) THEN
		
		CASE me.intCmd OF		
			JCL_CmdState.cCMD_Standby:
				me.StateMachine.intStateNext := JCL_CmdState.cSTA_StandbyBusy;			
		END_CASE
	END_IF

// --------------------------------------------------------------------------------------
// Exit action
	IF (me.StateMachine.intState<>me.StateMachine.intStateNext) THEN
		;
	END_IF
END_METHOD

{attribute 'object_name' := 'sta_CALIBRATIONBusy'}
METHOD PROTECTED sta_CALIBRATIONBusy : BOOL
VAR
	stNextCommand: T_JCL_Command;
	pNextCommand: POINTER TO T_JCL_Command;
END_VAR
// state implemetation
// --------------------------------------------------------------------------------------
// Entry action
	IF (me.StateMachine.intState<>me.StateMachine.intStateLastCycle) THEN
		me.StateMachine.intStateLastCycle := me.StateMachine.intState;
		
		// Simulation
		fbSimulationTimer.IN := FALSE;
		fbSimulationTimer.PT := T#5S;
		fbSimulationTimer(); // set time/reset timer
		fbSimulationTimer.IN := TRUE; // start timer
				
		IF CIf.SwCfg.bolSimulation THEN
			;
		ELSE
			// -----------------------------------------
			// Prepare telegram for standby
			// -----------------------------------------
			// Define header		
			stNextCommand.stHeader.uinMsgId := JCL_MsgId_Command;
			stNextCommand.stHeader.udiMsgSize := SIZEOF(T_JCL_Command) - SIZEOF(ST_Header);
			// Set DJM CMD
			stNextCommand.usiCommand := JCL_CMD_Calibration;
			// Push telegram to send buffer	
			pNextCommand := ADR(stNextCommand);
			p_fbTCP^.M_Push(paPushMsg := pNextCommand);	
		END_IF
		
	END_IF

// --------------------------------------------------------------------------------------
// Cyclic action
	IF (me.StateMachine.intState=me.StateMachine.intStateLastCycle) THEN
		
		// Simulation
		IF (CIf.SwCfg.bolSimulation) THEN
			fbSimulationTimer(); // simulation time
			IF (fbSimulationTimer.Q) THEN
				SIf.Cur.intJETState  := JCL_CmdState.cSTA_Calibration;
			END_IF
		END_IF	
	
		// Wait for feedback -> maintenance automatic done	
		IF (SIf.Cur.intJETState = JCL_CmdState.cSTA_Calibration) THEN
			me.StateMachine.intStateNext := JCL_CmdState.cSTA_Calibration;
		END_IF
		
	END_IF

// --------------------------------------------------------------------------------------
// Exit action
	IF (me.StateMachine.intState<>me.StateMachine.intStateNext) THEN
		;
	END_IF
END_METHOD

{attribute 'object_name' := 'sta_CLEANING'}
METHOD PROTECTED sta_CLEANING : BOOL
// state implemetation
// --------------------------------------------------------------------------------------
// Entry action
	IF (me.StateMachine.intState<>me.StateMachine.intStateLastCycle) THEN
		me.StateMachine.intStateLastCycle := me.StateMachine.intState;
		;
	END_IF

// --------------------------------------------------------------------------------------
// Cyclic action
	IF (me.StateMachine.intState=me.StateMachine.intStateLastCycle) THEN
		
		CASE me.intCmd OF	
			Base_PLC.cCMD_RUN:
				me.StateMachine.intStateNext := Base_PLC.cSTA_RUNBusy;	
			JCL_CmdState.cCMD_Standby:
				me.StateMachine.intStateNext := JCL_CmdState.cSTA_StandbyBusy;			
		END_CASE
	END_IF

// --------------------------------------------------------------------------------------
// Exit action
	IF (me.StateMachine.intState<>me.StateMachine.intStateNext) THEN
		;
	END_IF
END_METHOD

{attribute 'object_name' := 'sta_CLEANINGBusy'}
METHOD PROTECTED sta_CLEANINGBusy : BOOL
VAR
	stNextCommand: T_JCL_Command;
	pNextCommand: POINTER TO T_JCL_Command;
END_VAR
// state implemetation
// --------------------------------------------------------------------------------------
// Entry action
	IF (me.StateMachine.intState<>me.StateMachine.intStateLastCycle) THEN
		me.StateMachine.intStateLastCycle := me.StateMachine.intState;
		
		// Simulation
		fbSimulationTimer.IN := FALSE;
		fbSimulationTimer.PT := T#5S;
		fbSimulationTimer(); // set time/reset timer
		fbSimulationTimer.IN := TRUE; // start timer
				
		IF CIf.SwCfg.bolSimulation THEN
			;
		ELSE
			// -----------------------------------------
			// Prepare telegram for standby
			// -----------------------------------------
			// Define header		
			stNextCommand.stHeader.uinMsgId := JCL_MsgId_Command;
			stNextCommand.stHeader.udiMsgSize := SIZEOF(T_JCL_Command) - SIZEOF(ST_Header);
			// Set DJM CMD
			stNextCommand.usiCommand := JCL_CMD_CleanPrintHeads;
			// Push telegram to send buffer	
			pNextCommand := ADR(stNextCommand);
			p_fbTCP^.M_Push(paPushMsg := pNextCommand);	
		END_IF
		
	END_IF


// --------------------------------------------------------------------------------------
// Cyclic action
	IF (me.StateMachine.intState=me.StateMachine.intStateLastCycle) THEN
		
		// Simulation
		IF (CIf.SwCfg.bolSimulation) THEN
			fbSimulationTimer(); // simulation time
			IF (fbSimulationTimer.Q) THEN
				SIf.Cur.intJETState  := JCL_CmdState.cSTA_CleanPrintHeads;
			END_IF
		END_IF	
	
		// Wait for feedback -> maintenance automatic done	
		IF (SIf.Cur.intJETState = JCL_CmdState.cSTA_CleanPrintHeads) THEN
			me.StateMachine.intStateNext := JCL_CmdState.cSTA_CleanPrintHeads;
		END_IF
		
	END_IF

// --------------------------------------------------------------------------------------
// Exit action
	IF (me.StateMachine.intState<>me.StateMachine.intStateNext) THEN
		;
	END_IF
END_METHOD

{attribute 'object_name' := 'sta_CONNECTBusy'}
METHOD sta_CONNECTBusy : BOOL
VAR
	stNextCommand: T_JCL_Command;
	pNextCommand: POINTER TO T_JCL_Command;
END_VAR
// state implemetation
// --------------------------------------------------------------------------------------
// Entry action
	IF (me.StateMachine.intState<>me.StateMachine.intStateLastCycle) THEN
		me.StateMachine.intStateLastCycle := me.StateMachine.intState;
	
		// **********************************************************************************
		// This state will be executed one time after startup or after an error ack.
		// State open the TCP communication to jetter remote server to get the actual machine state
		// **********************************************************************************
		// Reset state 
		SIf.Cur.intJETState:= 0;
		
		// Connect to the jetter server
		pTCP_CIF^.Job.intACmd:= TCP_CmdState.cCMD_Connect;
		
		// Initialize sub state machine
		me.SubStateMachine.intStateNext:= JCL_CmdState.cSUB_WaitingForConnection;		
		me.SubStateMachine.intState:= me.SubStateMachine.intStateNext-1;
	END_IF

// --------------------------------------------------------------------------------------
// Cyclic action
	IF (me.StateMachine.intState=me.StateMachine.intStateLastCycle) THEN
		
		// -----------------------------------------------
		// Sub state machine handle 
		// -----------------------------------------------
		CASE me.SubStateMachine.intState OF
			
			JCL_CmdState.cSUB_WaitingForConnection:			
				// Wait for connection
				IF (pTCP_CIF^.Job.intState = TCP_CmdState.cSTA_Connect) THEN	
					// Request jetter states the first time after TCP client connected				
					THIS^.RequestState();		
					me.SubStateMachine.intStateNext:= JCL_CmdState.cSUB_WaitingForState;	
				END_IF
			
			JCL_CmdState.cSUB_WaitingForState:
				// Wait for first status msg 
				IF (SIf.Cur.intJETState > 0) THEN 
					me.SubStateMachine.intStateNext:= JCL_CmdState.cSUB_Done;
				END_IF	

			JCL_CmdState.cSUB_Done:
				// Change to the init state
				me.StateMachine.intStateNext := SIf.Cur.intJETState;
			
		END_CASE
			
	END_IF

// --------------------------------------------------------------------------------------
// Exit action
	IF (me.StateMachine.intState<>me.StateMachine.intStateNext) THEN
		;
	END_IF
END_METHOD

{attribute 'object_name' := 'sta_ERROR'}
METHOD PROTECTED sta_ERROR : BOOL
// state implemetation
// --------------------------------------------------------------------------------------
// Entry action
	IF (me.StateMachine.intState<>me.StateMachine.intStateLastCycle) THEN
		me.StateMachine.intStateHistory := me.StateMachine.intStateLastCycle; // -> possibillity to go back to state before error
		me.StateMachine.intStateLastCycle := me.StateMachine.intState;
		
	END_IF

// --------------------------------------------------------------------------------------
// Cyclic action
	IF (me.StateMachine.intState=me.StateMachine.intStateLastCycle) THEN
	
		// State Change Condition
		IF (CIf.Job.bolAlmReset = TRUE) THEN
			me.StateMachine.intStateNext := cSTA_ERRORQuit;
		END_IF
	END_IF

// --------------------------------------------------------------------------------------
// Exit action
	IF (me.StateMachine.intState<>me.StateMachine.intStateNext) THEN
		;
	END_IF
END_METHOD

{attribute 'object_name' := 'sta_ERRORQuit'}
METHOD PROTECTED sta_ERRORQuit : BOOL
// state implemetation
// --------------------------------------------------------------------------------------
// Entry action
	IF (me.StateMachine.intState<>me.StateMachine.intStateLastCycle) THEN
		me.StateMachine.intStateLastCycle := me.StateMachine.intState;
		
	END_IF

// --------------------------------------------------------------------------------------
// Cyclic action
	IF (me.StateMachine.intState=me.StateMachine.intStateLastCycle) THEN
		
		// evtl. wait time if reset of device is necessary and then decide to go to states or ERROR state
		IF (CIf.Job.bolAlmReset = TRUE) THEN
			CIf.Job.eMe_ActivAlmClass := E_AlmClass.NONE; // reset feedback channel for parent
			CIf.Job.bolAlmReset := FALSE;
		END_IF
		
		// State Change Condition
		IF (pTCP_CIF^.Job.bolAlmReset = FALSE) THEN
	
			// If the error was triggered because of an TCP connection problem to the server
			IF (bolServerConnectionError) AND (pTCP_CIF^.Job.eMe_ActivAlmClass = E_AlmClass.NONE) THEN
				bolServerConnectionError:= FALSE;
				// Try to reopen the connection to server
				me.StateMachine.intStateNext := JCL_CmdState.cSTA_ConnectBusy;
			END_IF
		
			CASE me.intCmd OF
				BASE_PLC.cCMD_OFF:
					me.StateMachine.intStateNext := BASE_PLC.cSTA_OFFBusy;
			END_CASE
			
		END_IF
	END_IF

// --------------------------------------------------------------------------------------
// Exit action
	IF (me.StateMachine.intState<>me.StateMachine.intStateNext) THEN
		;
	END_IF
END_METHOD

{attribute 'object_name' := 'sta_OFF'}
METHOD PROTECTED sta_OFF : BOOL
// state implemetation
// --------------------------------------------------------------------------------------
// Entry action
	IF (me.StateMachine.intState<>me.StateMachine.intStateLastCycle) THEN
		me.StateMachine.intStateLastCycle := me.StateMachine.intState;	
		;
	END_IF


// --------------------------------------------------------------------------------------
// Cyclic action
	IF (me.StateMachine.intState=me.StateMachine.intStateLastCycle) THEN
	
		CASE me.intCmd OF
			Base_PLC.cCMD_RUN: 				
				me.StateMachine.intStateNext := Base_PLC.cSTA_RUNBusy;	
			JCL_CmdState.cCMD_Standby: 				
				me.StateMachine.intStateNext := JCL_CmdState.cSTA_StandbyBusy;
			JCL_CmdState.cCMD_CleanPrintHeads: 				
				me.StateMachine.intStateNext := JCL_CmdState.cSTA_CleanPrintHeadsBusy;
		END_CASE
		
	END_IF


// --------------------------------------------------------------------------------------
// Exit action
	IF (me.StateMachine.intState<>me.StateMachine.intStateNext) THEN
		;
	END_IF
END_METHOD

{attribute 'object_name' := 'sta_OFFBusy'}
METHOD PROTECTED sta_OFFBusy : BOOL
VAR
	stNextCommand: T_JCL_Command;
	pNextCommand: POINTER TO T_JCL_Command;
END_VAR
// state implemetation
// --------------------------------------------------------------------------------------
// Entry action
IF (me.StateMachine.intState<>me.StateMachine.intStateLastCycle) THEN
	me.StateMachine.intStateLastCycle := me.StateMachine.intState;
	
	IF (CIf.SwCfg.bolSimulation) THEN 
		SIf.Cur.bolReadyForProduction:= TRUE;			
		SIf.Cur.bolRunning:= FALSE;		
		SIf.Cur.bolNeedsAttention:= FALSE;			
		SIf.Cur.bolError:= FALSE;			
		SIf.Cur.bolCleaningIncomplete:= FALSE;			
		SIf.Cur.bolIsLocalControlled:= FALSE;		
		SIf.Cur.bolIsRemoteControlled:= TRUE;
		SIf.Cur.intJETState := BASE_PLC.cSTA_OFF;
	ELSE 
		// -----------------------------------------
		// Prepare telegram for off
		// -----------------------------------------
		// Define header
		stNextCommand.stHeader.uinMsgId := JCL_MsgId_Command;
		stNextCommand.stHeader.udiMsgSize := SIZEOF(T_JCL_Command) - SIZEOF(ST_Header);
		// Set jetter CMD
		stNextCommand.usiCommand := JCL_CMD_Off;
		// Push telegram to send buffer
		pNextCommand := ADR(stNextCommand);
		p_fbTCP^.M_Push(paPushMsg := pNextCommand);	
	END_IF
	
END_IF

// --------------------------------------------------------------------------------------
// Cyclic action
IF (me.StateMachine.intState=me.StateMachine.intStateLastCycle) THEN
	
	// Wait for feedback -> OFF
	IF (SIf.Cur.intJETState = BASE_PLC.cSTA_OFF) THEN
		me.StateMachine.intStateNext := cSTA_OFF;
	END_IF
	
END_IF

// --------------------------------------------------------------------------------------
// Exit action
IF (me.StateMachine.intState<>me.StateMachine.intStateNext) THEN
	;
END_IF
END_METHOD

{attribute 'object_name' := 'sta_PON'}
METHOD PROTECTED sta_PON : BOOL
// state implemetation
// --------------------------------------------------------------------------------------
// Entry action
	IF (me.StateMachine.intState<>me.StateMachine.intStateLastCycle) THEN
		me.StateMachine.intStateLastCycle := me.StateMachine.intState;
		

		
	END_IF

// --------------------------------------------------------------------------------------
// Cyclic action
	IF (me.StateMachine.intState=me.StateMachine.intStateLastCycle) THEN	
		
		CASE me.intCmd OF
			cCMD_OFF: 				
				me.StateMachine.intStateNext := cSTA_OFFBusy;
			JCL_CmdState.cCMD_Standby:
				me.StateMachine.intStateNext := JCL_CmdState.cSTA_StandbyBusy;
			cCMD_Run:
				me.StateMachine.intStateNext := cSTA_RUNBusy;
		END_CASE
	
	END_IF
	
// --------------------------------------------------------------------------------------
// Exit action
	IF (me.StateMachine.intState<>me.StateMachine.intStateNext) THEN
		;
	END_IF
END_METHOD

{attribute 'object_name' := 'sta_PONBusy'}
METHOD PROTECTED sta_PONBusy : BOOL
VAR
	stNextCommand: T_JCL_Command;
	pNextCommand: POINTER TO T_JCL_Command;
END_VAR
// state implemetation
// --------------------------------------------------------------------------------------
// Entry action
IF (me.StateMachine.intState<>me.StateMachine.intStateLastCycle) THEN
	me.StateMachine.intStateLastCycle := me.StateMachine.intState;
	
	IF NOT (CIf.SwCfg.bolSimulation) THEN
		// If the socket is already connected, trigger a reconnet.
		IF (pTCP_CIF^.Job.intState = TCP_CmdState.cSTA_Connect) OR (pTCP_CIF^.Job.intState = Base_PLC.cSTA_ERROR) THEN
			// Initialize sub state machine
			me.SubStateMachine.intStateNext:= JCL_CmdState.cSUB_WaitingSocketClosed;		
			me.SubStateMachine.intState:= me.SubStateMachine.intStateNext-1;
			// Connect to jetter server
			pTCP_CIF^.Job.intACmd:= TCP_CmdState.cCMD_Close;	
		ELSE		
			// Initialize sub state machine
			me.SubStateMachine.intStateNext:= JCL_CmdState.cSUB_WaitingForConnection;		
			me.SubStateMachine.intState:= me.SubStateMachine.intStateNext-1;
			// Connect to jetter server
			pTCP_CIF^.Job.intACmd:= TCP_CmdState.cCMD_Connect;	
		END_IF
	ELSE
		SIf.Cur.bolReadyForProduction:= TRUE;			
		SIf.Cur.bolRunning:= FALSE;		
		SIf.Cur.bolNeedsAttention:= FALSE;			
		SIf.Cur.bolError:= FALSE;			
		SIf.Cur.bolCleaningIncomplete:= FALSE;			
		SIf.Cur.bolIsLocalControlled:= FALSE;		
		SIf.Cur.bolIsRemoteControlled:= TRUE;
		SIf.Cur.intJETState := BASE_PLC.cSTA_PON;
	END_IF
	
END_IF

// --------------------------------------------------------------------------------------
// Cyclic action
IF (me.StateMachine.intState=me.StateMachine.intStateLastCycle) THEN
	
	CASE me.SubStateMachine.intState OF
			
		JCL_CmdState.cSUB_WaitingSocketClosed:	
			IF (CIf.SwCfg.bolSimulation) THEN
				me.SubStateMachine.intStateNext:= JCL_CmdState.cSUB_WaitingForConnection;	
			ELSE							
				// Wait for socket closed
				IF (pTCP_CIF^.Job.intState = TCP_CmdState.cSTA_Close) THEN			
					me.SubStateMachine.intStateNext:= JCL_CmdState.cSUB_WaitingForConnection;	
				END_IF		
			END_IF
	
		JCL_CmdState.cSUB_WaitingForConnection:		
			IF (CIf.SwCfg.bolSimulation) THEN
				me.SubStateMachine.intStateNext:= JCL_CmdState.cSUB_SendPon;	
			ELSE							
				// Connect to jetter server
				pTCP_CIF^.Job.intACmd:= TCP_CmdState.cCMD_Connect;	
					
				// Wait for connection
				IF (pTCP_CIF^.Job.intState = TCP_CmdState.cSTA_Connect) THEN			
					me.SubStateMachine.intStateNext:= JCL_CmdState.cSUB_SendPon;	
				END_IF		
			END_IF
					
		JCL_CmdState.cSUB_SendPon:	
			// Prepare telegram for PON
			// -----------------------------------------
			// Define header
			stNextCommand.stHeader.uinMsgId := JCL_MsgId_Command;
			stNextCommand.stHeader.udiMsgSize := SIZEOF(T_JCL_Command) - SIZEOF(ST_Header);
			// Set jetter CMD
			stNextCommand.usiCommand := JCL_CMD_PowerOn;
			// Push telegram to send buffer
			pNextCommand := ADR(stNextCommand);
			p_fbTCP^.M_Push(paPushMsg := pNextCommand);	
			me.SubStateMachine.intStateNext:= JCL_CmdState.cSUB_Done;	
					
		JCL_CmdState.cSUB_Done:
			// ... do nothing
	
	END_CASE

	// Wait for feedback -> PON
	IF (SIf.Cur.intJETState = BASE_PLC.cSTA_PON) OR (SIf.Cur.intJETState = BASE_PLC.cSTA_OFF) THEN
		me.StateMachine.intStateNext := cSTA_PON;
	END_IF
	
END_IF

// --------------------------------------------------------------------------------------
// Exit action
IF (me.StateMachine.intState<>me.StateMachine.intStateNext) THEN
	;
END_IF
END_METHOD

{attribute 'object_name' := 'sta_RUN'}
METHOD PROTECTED sta_RUN : BOOL
// state implemetation
// --------------------------------------------------------------------------------------
// Entry action
	IF (me.StateMachine.intState<>me.StateMachine.intStateLastCycle) THEN
		me.StateMachine.intStateLastCycle := me.StateMachine.intState;
		
	END_IF

// --------------------------------------------------------------------------------------
// Cyclic action
	IF (me.StateMachine.intState=me.StateMachine.intStateLastCycle) THEN
		
		CASE me.intCmd OF
			Base_PLC.cCMD_RUN:
				me.StateMachine.intStateNext := Base_PLC.cSTA_RUNBusy;	
			JCL_CmdState.cCMD_CleanPrintHeads:
				me.StateMachine.intStateNext := JCL_CmdState.cSTA_CleanPrintHeadsBusy;
			JCL_CmdState.cCMD_Standby:
				me.StateMachine.intStateNext := JCL_CmdState.cSTA_StandbyBusy;
		END_CASE
		
	END_IF
	

// --------------------------------------------------------------------------------------
// Exit action
	IF (me.StateMachine.intState<>me.StateMachine.intStateNext) THEN
		;
	END_IF
END_METHOD

{attribute 'object_name' := 'sta_RUNBusy'}
METHOD PROTECTED sta_RUNBusy : BOOL
VAR
	stNextCommand: T_JCL_Command;
	pNextCommand: POINTER TO T_JCL_Command;
END_VAR
// state implemetation
// --------------------------------------------------------------------------------------
// Entry action
	IF (me.StateMachine.intState<>me.StateMachine.intStateLastCycle) THEN
		me.StateMachine.intStateLastCycle := me.StateMachine.intState;
		
		IF CIf.SwCfg.bolSimulation THEN
			SIf.Cur.bolReadyForProduction:= TRUE;			
			SIf.Cur.bolRunning:= TRUE;		
			SIf.Cur.bolNeedsAttention:= FALSE;			
			SIf.Cur.bolError:= FALSE;			
			SIf.Cur.bolCleaningIncomplete:= FALSE;			
			SIf.Cur.bolIsLocalControlled:= FALSE;		
			SIf.Cur.bolIsRemoteControlled:= TRUE;
			SIf.Cur.intJETState := cSTA_RUN;
		ELSE
			// -----------------------------------------
			// Prepare telegram for run
			// -----------------------------------------
			// Define header
			stNextCommand.stHeader.uinMsgId := JCL_MsgId_Command;
			stNextCommand.stHeader.udiMsgSize := SIZEOF(T_JCL_Command) - SIZEOF(ST_Header);
			// Set jetter CMD
			stNextCommand.usiCommand := JCL_CMD_Run;
			// Push telegram to send buffer
			pNextCommand := ADR(stNextCommand);
			p_fbTCP^.M_Push(paPushMsg := pNextCommand);
		END_IF
			 
	END_IF


// --------------------------------------------------------------------------------------
// Cyclic action
	IF (me.StateMachine.intState=me.StateMachine.intStateLastCycle) THEN
		
		// Wait for feedback -> RUN
		IF (SIf.Cur.intJETState = cSTA_RUN) THEN
			me.StateMachine.intStateNext := BASE_PLC.cSTA_RUN;
		END_IF
		
	END_IF

// --------------------------------------------------------------------------------------
// Exit action
	IF (me.StateMachine.intState<>me.StateMachine.intStateNext) THEN
		;
	END_IF
END_METHOD

{attribute 'object_name' := 'sta_STANDBY'}
METHOD PROTECTED sta_STANDBY : BOOL
// state implemetation
// --------------------------------------------------------------------------------------
// Entry action
	IF (me.StateMachine.intState<>me.StateMachine.intStateLastCycle) THEN
		me.StateMachine.intStateLastCycle := me.StateMachine.intState;
		;
	END_IF

// --------------------------------------------------------------------------------------
// Cyclic action
	IF (me.StateMachine.intState=me.StateMachine.intStateLastCycle) THEN
		
		CASE me.intCmd OF
			BASE_PLC.cCMD_RUN:
				me.StateMachine.intStateNext := BASE_PLC.cSTA_RUNBusy;
			JCL_CmdState.cCMD_Standby:
				me.StateMachine.intStateNext := JCL_CmdState.cSTA_StandbyBusy;
			JCL_CmdState.cCMD_CleanPrintHeads: 				
				me.StateMachine.intStateNext := JCL_CmdState.cSTA_CleanPrintHeadsBusy;
			JCL_CmdState.cCMD_Calibration: 				
				me.StateMachine.intStateNext := JCL_CmdState.cSTA_CalibrationBusy;	
		END_CASE
	END_IF

// --------------------------------------------------------------------------------------
// Exit action
	IF (me.StateMachine.intState<>me.StateMachine.intStateNext) THEN
		;
	END_IF
END_METHOD

{attribute 'object_name' := 'sta_STANDBYBusy'}
METHOD PROTECTED sta_STANDBYBusy : BOOL
VAR
	stNextCommand: T_JCL_Command;
	pNextCommand: POINTER TO T_JCL_Command;
END_VAR
// state implemetation
// --------------------------------------------------------------------------------------
// Entry action
	IF (me.StateMachine.intState<>me.StateMachine.intStateLastCycle) THEN
		me.StateMachine.intStateLastCycle := me.StateMachine.intState;
		
		// Simulation
		fbSimulationTimer.IN := FALSE;
		fbSimulationTimer.PT := T#5S;
		fbSimulationTimer(); // set time/reset timer
		fbSimulationTimer.IN := TRUE; // start timer
				
		IF CIf.SwCfg.bolSimulation THEN
			;
		ELSE
			// -----------------------------------------
			// Prepare telegram for standby
			// -----------------------------------------
			// Define header		
			stNextCommand.stHeader.uinMsgId := JCL_MsgId_Command;
			stNextCommand.stHeader.udiMsgSize := SIZEOF(T_JCL_Command) - SIZEOF(ST_Header);
			// Set DJM CMD
			stNextCommand.usiCommand := JCL_CMD_Standby;
			// Push telegram to send buffer	
			pNextCommand := ADR(stNextCommand);
			p_fbTCP^.M_Push(paPushMsg := pNextCommand);	
		END_IF
		
	END_IF


// --------------------------------------------------------------------------------------
// Cyclic action
	IF (me.StateMachine.intState=me.StateMachine.intStateLastCycle) THEN
		
		// Simulation
		IF (CIf.SwCfg.bolSimulation) THEN
			fbSimulationTimer(); // simulation time
			IF (fbSimulationTimer.Q) THEN
				SIf.Cur.bolReadyForProduction:= TRUE;			
				SIf.Cur.bolRunning:= TRUE;		
				SIf.Cur.bolNeedsAttention:= FALSE;			
				SIf.Cur.bolError:= FALSE;			
				SIf.Cur.bolCleaningIncomplete:= FALSE;			
				SIf.Cur.bolIsLocalControlled:= FALSE;		
				SIf.Cur.bolIsRemoteControlled:= TRUE;
				SIf.Cur.intJETState  := JCL_CmdState.cSTA_Standby;
			END_IF
		END_IF	
	
		// Wait for feedback -> standby	
		IF (SIf.Cur.intJETState  = JCL_CmdState.cSTA_Standby) THEN
			me.StateMachine.intStateNext := JCL_CmdState.cSTA_Standby;
		END_IF
		
	END_IF

// --------------------------------------------------------------------------------------
// Exit action
	IF (me.StateMachine.intState<>me.StateMachine.intStateNext) THEN
		;
	END_IF
END_METHOD

{attribute 'object_name' := 'StateMachine'}
METHOD PROTECTED StateMachine : BOOL
SUPER^.StateMachine();

// main statemachine of base controller
CASE me.StateMachine.intState OF
	JCL_CmdState.cSTA_ConnectBusy: 
        THIS^.sta_CONNECTBusy();
	cSTA_RUNBusy: 
        THIS^.sta_RUNBusy();
	cSTA_RUN: 
        THIS^.sta_RUN();
	JCL_CmdState.cSTA_StandbyBusy: 
        THIS^.sta_STANDBYBusy();
	JCL_CmdState.cSTA_Standby: 
        THIS^.sta_STANDBY();	
	JCL_CmdState.cSTA_CleanPrintHeadsBusy: 
        THIS^.sta_CLEANINGBusy();
	JCL_CmdState.cSTA_CleanPrintHeads: 
        THIS^.sta_CLEANING();	
	JCL_CmdState.cSTA_CalibrationBusy:
		THIS^.sta_CALIBRATIONBusy();
	JCL_CmdState.cSTA_Calibration:
		THIS^.sta_CALIBRATION();
END_CASE
END_METHOD

PROPERTY TCP : POINTER TO FB_TCP
GET
TCP := p_fbTCP;
END_GET
SET
p_fbTCP := TCP;
END_SET
END_PROPERTY

END_FUNCTION_BLOCK

// POUs/Controller/Utility/LookupTable/FB_LookupTable
FUNCTION_BLOCK FB_LookupTable
VAR_INPUT
	iAddKey: INT;
	iAddValue: INT;
	iLookupKey: INT;
	iLookupValue: INT;
END_VAR
VAR_OUTPUT
	/// number of elements in Table
	iCount: INT;
	bOK: BOOL;
	iFoundValue: INT;
	iFoundKey: INT;
END_VAR
VAR
	aiKeys: ARRAY[0..MaxLookupSize] OF INT;
	aiValues: ARRAY[0..MaxLookupSize] OF INT;
	ii: INT;
	bDone: BOOL;
END_VAR

(* 
	This is a very slow lookup table! do not use for big amounts of data
*)

ACTION A_Add:
IF (iAddKey = 0) OR (iCount = MaxLookupSize) THEN
	bOK := 0; 
	RETURN;
END_IF
bDone := 0;

FOR ii := 0 TO MaxLookupSize BY 1 DO // see if key already exists
	IF ( iAddKey = aiKeys[ii] ) THEN // overwrite old element
		aiValues[ii] := iAddValue;
		bOK := 1;
		bDone := 1;
		RETURN;
	END_IF
END_FOR

// add new entry
// find first unused element in table
FOR ii := 0 TO MaxLookupSize BY 1 DO
	IF aiKeys[ii] = 0 THEN
		aiKeys[ii] := iAddKey;
		aiValues[ii] := iAddValue;
		iCount := iCount +1;
		bOK := 1;
		RETURN;
	END_IF
END_FOR
END_ACTION

ACTION A_LookupByKey:
bOK := 0;

FOR ii := 0 TO MaxLookupSize BY 1 DO
	IF iLookupKey = aiKeys[ii] THEN // found it
		iFoundValue := aiValues[ii];
		bOK := 1;
		RETURN;
	END_IF
END_FOR
END_ACTION

ACTION A_LookupByValue:
// will only find the first key associated with the value
bOK := 0;

FOR ii := 0 TO MaxLookupSize BY 1 DO
	IF iLookupValue = aiValues[ii] THEN // found it
		iFoundKey := aiKeys[ii];
		bOK := 1;
		RETURN;
	END_IF
END_FOR
END_ACTION

ACTION A_RemoveKey:
bOK := 0;

FOR ii := 0 TO MaxLookupSize BY 1 DO
	IF iLookupKey = aiKeys[ii] THEN // found it
		aiKeys[ii] := 0;
		aiValues[ii] := 0;
		bOK := 1;
		RETURN;
	END_IF
END_FOR
END_ACTION

ACTION A_Reset:
FOR ii := 0 TO MaxLookupSize BY 1 DO
	aiKeys[ii] := 0;
	aiValues[ii] := 0;
END_FOR
bOK := 1;
END_ACTION

END_FUNCTION_BLOCK

// POUs/Controller/Lvl0/RAX(Rotative Axis)/FB_RAX
FUNCTION_BLOCK FB_RAX EXTENDS FB_CtrlBase
VAR_INPUT
	In_pAD_SIf: POINTER TO T_POD;
END_VAR
VAR
	/// Specific interface struct for public access
	SIf: T_Ctrl_SIf_RAX;
	/// internal variables
	ii: UINT;
END_VAR
VAR CONSTANT
	/// ctrl specific substates definitions
	cSUB_INITIALIZED: INT := 500;
	cSUB_WriteSW: INT := 501;
	cSUB_Home: INT := 502;
	cSUB_MoveToInitPos: INT := 503;
	cSUB_Finished: INT := 504;
END_VAR

(*__________________________________________________________________________________________________
¦	
¦	Vistaprint Schweiz GmbH
¦	CH - 8401 Winterthur
¦
¦	www.vistaprint.ch - info@vistaprint.ch
¦___________________________________________________________________________________________________

Function desription:
Rotary axis controller based on Deg unit system.

- position POS moved with absolute positioning
- nc settings base unit in Degree!!
- REL_POS -> relative positioning for single command

History:
Version		Date			Author		Comment
---------------------------------------------------------------------------------------------------
0.00.1		12.09.2014		AVME/KVO	Start history
0.00.2		22.09.2014		AVME/MRU	Copy of LAX, renamed to RAX, changed mm to Degree,
										Added Turn

_______________________________________________________________________________________________*)

IF (me.bolActivate) AND (In_pAD_SIf<>0) THEN // cyclic call enabled
	
	IF (CIf.Info.bolInitDone=FALSE) THEN // first cycle -> init
		CtrlInit();
		CIf.Info.bolInitDone := TRUE;
	ELSE
		CycleStartDuty();
	
		Always();
		
		StateMachine();
		
		CycleEndDuty();
	END_IF
END_IF;

{attribute 'object_name' := 'Always'}
METHOD PROTECTED Always : BOOL
SUPER^.Always();

// ----------------------------------------------------------------------------------
// cyclic actions outside of statemachine
IF (me.StateMachine.intState<>cSTA_SINGLE_ANSWER) THEN
	
	// always
	SIf.Cur.dinPosition_0_1deg := LREAL_TO_DINT(In_pAD_SIf^.stMove.lreActPos)*10;
	SIf.Cur.dinModPosition_0_1deg := LREAL_TO_DINT(In_pAD_SIf^.stMove.lreActModPos)*10;
	SIf.Cur.dinSpeed_0_1deg_s := LREAL_TO_DINT(In_pAD_SIf^.stMove.lreActVel)*10;
	SIf.Cur.dinTorque_0_1Nm := LREAL_TO_DINT(In_pAD_SIf^.stMove.lreActTorque)*10;
	SIf.Cur.bol_di1 := In_pAD_SIf^.stStatus.stDigIn.bol_SI0;
	SIf.Cur.bol_di2 := In_pAD_SIf^.stStatus.stDigIn.bol_SI1;
	SIf.Cur.bol_di3 := In_pAD_SIf^.stStatus.stDigIn.bol_SI2;
	SIf.Cur.bol_di4 := In_pAD_SIf^.stStatus.stDigIn.bol_SI3; // used for homing.....

	// info message 'software limit reached'
	IF ((In_pAD_SIf^.stStatus.bolNegSWSwitch) OR (In_pAD_SIf^.stStatus.bolPosSWSwitch)) THEN 
		IF (SIf.Alm[E_ALM_RAX.SwLimit].bol=FALSE)THEN
			// 'software limit reached';
			pfbAlarmCtrl^.setAlarm(CIf.Info.intCtrlId,E_ALM_RAX.SwLimit,0,ADR(SIf.Alm),E_AlmState.SET,CIf.Job.eMe_ActivAlmClass);
			SIf.Alm[E_ALM_RAX.SwLimit].bol:= TRUE;
		END_IF;
	ELSE
		IF (SIf.Alm[E_ALM_RAX.SwLimit].bol) THEN
			pfbAlarmCtrl^.setAlarm(CIf.Info.intCtrlId,4,0,ADR(SIf.Alm),E_AlmState.CLR,CIf.Job.eMe_ActivAlmClass);
			SIf.Alm[E_ALM_RAX.SwLimit].bol:= FALSE;
		END_IF
	END_IF
	
	//------------------------------------------------------------------------------------------------------------------------------------
	// set parameter
	// in Manual set % speed to 100% for single cmd's
	IF (CIf.Job.eMode=E_Mode.MANU) THEN
		SIf.Par.dinSpeed_per := 100;
		SIf.Par.dinAcc_per := 100;
		SIf.Par.dinDec_per := 100;
	END_IF	
	
	In_pAD_SIf^.stMove.lreSetSpeed := fSetPar(SIf.Par.dinSpeed_0_1deg_s,SIf.Par.dinSpeed_per);
	In_pAD_SIf^.stMove.lreSetAcc := fSetPar(SIf.Par.dintAccDec_0_1deg_s2,SIf.Par.dinAcc_per);
	In_pAD_SIf^.stMove.lreSetDec := fSetPar(SIf.Par.dintAccDec_0_1deg_s2,SIf.Par.dinDec_per);
	IF (SIf.Par.dinSetDecFast_0_1deg_s2>0) THEN
		In_pAD_SIf^.stMove.lreSetDecFast := DINT_TO_LREAL(SIf.Par.dinSetDecFast_0_1deg_s2)/10.0;
	ELSE
		In_pAD_SIf^.stMove.lreSetDecFast := In_pAD_SIf^.stMove.lreSetDec;
	END_IF
	In_pAD_SIf^.stCfg.bolSimulation := CIf.SwCfg.bolSimulation;
	
	// ----------------------------------------------------------------------------------
	// Conditions Always
	IF (me.StateMachine.intState>cSTA_PON) THEN	
		IF ((In_pAD_SIf^.stErr.bolErrorActive) AND (me.StateMachine.intState<>cSTA_ERROR) AND (me.StateMachine.intState<>cSTA_ERRORQuit)) THEN
			// detect drive error
			me.StateMachine.intStateNext := cSTA_ERROR;
		END_IF
	END_IF
END_IF
END_METHOD

PROPERTY PUBLIC CtrlSIf : POINTER TO T_Ctrl_SIf_RAX
GET
CtrlSIf := ADR(SIf);
END_GET
END_PROPERTY

{attribute 'object_name' := 'FB_init'}
METHOD FB_init : BOOL
VAR_INPUT
	///if TRUE, the retain variables are initialized (warm start / cold start)
	bInitRetains: BOOL;
	///if TRUE, the instance afterwards gets moved into the copy code (online change)
	bInCopyCode: BOOL;
END_VAR
VAR
	udiTaskCnt: UDINT;
END_VAR
//------------------------------------------------------------------------------------------------------------------------
// to manually change in new FUB implementation!!!
// define valid commands for this controller
FOR ii:= 0 TO (SIZEOF(CIf.Job.aCmdList)/SIZEOF(CIf.Job.aCmdList[0])-1) BY 1 DO
	IF (CIf.Job.aCmdList[ii].intCmd=cCMD_INITIALIZED) THEN
		// found first empty array element
		EXIT;
	END_IF
END_FOR
CIf.Job.aCmdList[ii].intCmd := cCMD_INIT;
CIf.Job.aCmdList[ii].strName := 'Init'; 
CIf.Job.aCmdList[ii].bolAvailable := TRUE;
ii := ii +1;
CIf.Job.aCmdList[ii].intCmd := RAX_CmdState.cCMD_POS;
CIf.Job.aCmdList[ii].strName := 'Position absolute';
CIf.Job.aCmdList[ii].bolAvailable := TRUE;
ii := ii +1;
CIf.Job.aCmdList[ii].intCmd := RAX_CmdState.cCMD_JOG_NEG;
CIf.Job.aCmdList[ii].strName := 'jogging negativ direction';
CIf.Job.aCmdList[ii].bolAvailable := TRUE;
ii := ii +1;
CIf.Job.aCmdList[ii].intCmd := RAX_CmdState.cCMD_JOG_POS;
CIf.Job.aCmdList[ii].strName := 'jogging positive direction';
CIf.Job.aCmdList[ii].bolAvailable := TRUE;
ii := ii +1;
CIf.Job.aCmdList[ii].intCmd := RAX_CmdState.cCMD_HOME;
CIf.Job.aCmdList[ii].strName := 'Home';
CIf.Job.aCmdList[ii].bolAvailable := TRUE;
ii := ii +1;
CIf.Job.aCmdList[ii].intCmd := RAX_CmdState.cCMD_REL_POS;
CIf.Job.aCmdList[ii].strName := 'Relative move';
CIf.Job.aCmdList[ii].bolAvailable := TRUE;
ii := ii +1;
CIf.Job.aCmdList[ii].intCmd := RAX_CmdState.cCMD_TURN;
CIf.Job.aCmdList[ii].strName := 'Turn';
CIf.Job.aCmdList[ii].bolAvailable := TRUE;
ii := ii +1;

// set name of class/typ
CIf.Info.strType := 'FB_RAX';
CIf.Info.strFullName := 'Rotative Axis';

// set alarm class
SIf.Alm[E_ALM_RAX.GeneralDrive].eAlmClass := E_AlmClass.OFF;
SIf.Alm[E_ALM_RAX.GeneralDrive].strText := 'general drive failure -> info number'; 
SIf.Alm[E_ALM_RAX.GeneralNc].eAlmClass := E_AlmClass.OFF;
SIf.Alm[E_ALM_RAX.GeneralNc].strText := 'general nc failure -> info number';
SIf.Alm[E_ALM_RAX.SwLimit].eAlmClass := E_AlmClass.INFO;
SIf.Alm[E_ALM_RAX.SwLimit].strText := 'software limit reached';
SIf.Alm[E_ALM_RAX.NegHwLimit].eAlmClass := E_AlmClass.OFF;
SIf.Alm[E_ALM_RAX.NegHwLimit].strText := 'neg. hardware switch detected';
SIf.Alm[E_ALM_RAX.PosHwLimit].eAlmClass := E_AlmClass.OFF;
SIf.Alm[E_ALM_RAX.PosHwLimit].strText := 'pos. hardware switch detected';
SIf.Alm[E_ALM_RAX.InterlockNegMove].eAlmClass := E_AlmClass.EOFF;
SIf.Alm[E_ALM_RAX.InterlockNegMove].strText := 'interlock neg. movement - movement stopped';
SIf.Alm[E_ALM_RAX.InterlockPosMove].eAlmClass := E_AlmClass.EOFF;
SIf.Alm[E_ALM_RAX.InterlockPosMove].strText := 'interlock pos. movement  - movement stopped';
SIf.Alm[E_ALM_RAX.GeneralMCFUB].eAlmClass := E_AlmClass.STOP;
SIf.Alm[E_ALM_RAX.GeneralMCFUB].strText := 'MC fub error -> info number';

//*******************************************************************************
// initial values
//*******************************************************************************

// software configuration
CIf.SwCfg.bolExist := TRUE;
CIf.SwCfg.bolSimulation := FALSE;

// cfg
//SIf.Cfg.eHomingMode := MC_HomingMode.MC_Direct;
SIf.Cfg.eHomingMode := MC_HomingMode.MC_DefaultHoming;
SIf.Cfg.lreShortestWayWindow_deg := 20.0; //20.0°

// parmeter
SIf.Par.dinHomeOffset_0_1deg := -900;
SIf.Par.dinPos_0_1deg := 0;
SIf.Par.dinRelDist_0_1deg := 10;
SIf.Par.dinPositionInit_0_1deg := 0;
SIf.Par.dintAccDec_0_1deg_s2 := 4000;
SIf.Par.dinAcc_per := 100;
SIf.Par.dinDec_per := 100;
SIf.Par.dinSetDecFast_0_1deg_s2 := 4000;
SIf.Par.dinSpeed_0_1deg_s := 200;
SIf.Par.dinSpeed_per := 200;
SIf.Par.dinSWLimitNeg_0_1deg := 0;
SIf.Par.dinSWLimitPos_0_1deg := 360;
END_METHOD

{attribute 'object_name' := 'getCmdState'}
METHOD PROTECTED getCmdState : STRING
VAR_INPUT
	intCmdState: INT;
	bolState: BOOL;
END_VAR
getCmdState := SUPER^.getCmdState(intCmdState:=intCmdState,bolState:=bolState); // get global/base defined cmds/states
IF (getCmdState='') THEN // global not defined get local
	// get string cmd/state string information in runtime
	IF (bolState=FALSE) THEN
		// cmd's
		CASE intCmdState OF
			RAX_CmdState.cCMD_HOME: 
				getCmdState := 'cCMD_HOME';
			RAX_CmdState.cCMD_POS: 
				getCmdState := 'cCMD_POS';
			RAX_CmdState.cCMD_JOG_NEG: 
				getCmdState := 'cCMD_JOG_NEG';
			RAX_CmdState.cCMD_JOG_POS: 
				getCmdState := 'cCMD_JOG_POS';
			RAX_CmdState.cCMD_REL_POS: 
				getCmdState := 'cCMD_REL_POS';
			RAX_CmdState.cCMD_TURN: 
				getCmdState := 'cCMD_TURN';
		ELSE
				getCmdState := 'not defined';
		END_CASE;
	ELSE
	
	// cmd's
		CASE intCmdState OF
			RAX_CmdState.cSTA_POSBusy: 
				getCmdState := 'cSTA_POSBusy';
			RAX_CmdState.cSTA_POS: 
				getCmdState := 'cSTA_POS';
			RAX_CmdState.cSTA_JOG_NEG: 
				getCmdState := 'cSTA_JOG_NEG';
			RAX_CmdState.cSTA_JOG_POS: 
				getCmdState := 'cSTA_JOG_POS';
			RAX_CmdState.cSTA_REL_POSBusy: 
				getCmdState := 'cSTA_REL_POSBusy';
			RAX_CmdState.cSTA_REL_POS: 
				getCmdState := 'cSTA_REL_POS';
			RAX_CmdState.cSTA_TURNBusy: 
				getCmdState := 'cSTA_TURNBusy';
			RAX_CmdState.cSTA_TURN: 
				getCmdState := 'cSTA_TURN';			
			cSUB_WriteSW: 
				getCmdState := 'cSUB_WriteSW';
			cSUB_Home: 
				getCmdState := 'cSUB_Home';
			cSUB_MoveToInitPos: 
				getCmdState := 'cSUB_MoveToInitPos';
			cSUB_Finished: 
				getCmdState := 'cSUB_Finished';
			cSUB_INITIALIZED:
				getCmdState := 'cSUB_INITIALIZED';
		ELSE
				getCmdState := 'not defined';
		END_CASE;
	END_IF
END_IF
END_METHOD

{attribute 'object_name' := 'getDirection'}
METHOD PROTECTED getDirection : MC_Direction
VAR_INPUT
	dinActualPosition: DINT;
	lreSetPosition: LREAL;
END_VAR
VAR
	Direction: MC_Direction;
	lreActualPosition: LREAL;
END_VAR
Direction := MC_Positive_Direction;	// MC_Shortest_Way, MC_Negative_Direction, 
lreActualPosition := DINT_TO_LREAL(dinActualPosition)/10.0;
IF (ABS(ABS(lreActualPosition) - ABS(lreSetPosition)) <= SIf.Cfg.lreShortestWayWindow_deg) THEN
	Direction := MC_Shortest_Way;
ELSIF (lreActualPosition < 0) THEN
	Direction := MC_Negative_Direction;
END_IF;

getDirection := Direction;
END_METHOD

{attribute 'object_name' := 'IoOutBridge'}
METHOD PROTECTED IoOutBridge : BOOL
// digitale and analoge inputs read from hardware or forcing
IF (CIf.SwCfg.bolSimulation = FALSE) THEN
	// check interlocks to prevent damages
	IF (CIf.Job.bolIlkOverwrite=FALSE) THEN
		IF (SIf.Ilk.bolMovePos) AND (In_pAD_SIf^.stStatus.bolCtrlOn)  AND ((In_pAD_SIf^.intCmd=cPOD_CMD_POS_JOG) OR (In_pAD_SIf^.intCmd=cPOD_CMD_POS_MOVE) OR
			((In_pAD_SIf^.stMove.lreSetPos > In_pAD_SIf^.stMove.lreActPos) AND (In_pAD_SIf^.intCmd=cPOD_CMD_ABS_MOVE)) OR
			((In_pAD_SIf^.intCmd=cPOD_CMD_REL_MOVE) AND (In_pAD_SIf^.stMove.lreSetPos>0)) OR (SIf.Cur.dinSpeed_0_1deg_s>5)  )THEN	
			// SIf.Alm[8].strText := 'interlock pos. movement  - movement stopped';
			pfbAlarmCtrl^.setAlarm(CIf.Info.intCtrlId,E_ALM_RAX.InterlockPosMove,0,ADR(SIf.Alm),E_AlmState.RST,CIf.Job.eMe_ActivAlmClass);
			In_pAD_SIf^.intCmd:=cPOD_CMD_EMCY_STOP_CTRL_OFF;
		END_IF
		IF (SIf.Ilk.bolMoveNeg) AND (In_pAD_SIf^.stStatus.bolCtrlOn)  AND ((In_pAD_SIf^.intCmd=cPOD_CMD_NEG_JOG) OR (In_pAD_SIf^.intCmd=cPOD_CMD_NEG_MOVE) OR
		 	(In_pAD_SIf^.intCmd=cPOD_CMD_HOME) OR
			((In_pAD_SIf^.stMove.lreSetPos < In_pAD_SIf^.stMove.lreActPos) AND (In_pAD_SIf^.intCmd=cPOD_CMD_ABS_MOVE)) OR
			((In_pAD_SIf^.intCmd=cPOD_CMD_REL_MOVE) AND (In_pAD_SIf^.stMove.lreSetPos<0)) OR (SIf.Cur.dinSpeed_0_1deg_s<-5)  )THEN		
			// 'interlock neg. movement - movement stopped';
			pfbAlarmCtrl^.setAlarm(CIf.Info.intCtrlId,E_ALM_RAX.InterlockNegMove,0,ADR(SIf.Alm),E_AlmState.RST,CIf.Job.eMe_ActivAlmClass);
			In_pAD_SIf^.intCmd:=cPOD_CMD_EMCY_STOP_CTRL_OFF;
		END_IF	
	END_IF

END_IF
END_METHOD

{attribute 'object_name' := 'sta_EOFF'}
METHOD PROTECTED sta_EOFF : BOOL
// state implemetation
//--------------------------------------------------------------------------------------
// Entry action
	IF (me.StateMachine.intState<>me.StateMachine.intStateLastCycle) THEN
		me.StateMachine.intStateLastCycle := me.StateMachine.intState;
		
	END_IF


